C03630=1120.994,-41.227,-48.761,179.607,5.616,149.108
C03631=1120.989,-40.977,-48.773,179.608,5.621,149.109
C03632=1120.983,-40.727,-48.785,179.609,5.626,149.109
C03633=1120.979,-40.477,-48.796,179.611,5.631,149.110
C03634=1120.973,-40.227,-48.808,179.612,5.637,149.111
C03635=1120.969,-39.978,-48.819,179.613,5.642,149.112
C03636=1120.963,-39.729,-48.831,179.614,5.647,149.113
C03637=1120.957,-39.479,-48.843,179.615,5.652,149.113
C03638=1120.952,-39.229,-48.854,179.616,5.658,149.114
C03639=1120.947,-38.979,-48.866,179.618,5.663,149.115
C03640=1120.942,-38.729,-48.878,179.618,5.668,149.116
C03641=1120.937,-38.480,-48.890,179.620,5.673,149.116
C03642=1120.932,-38.230,-48.902,179.620,5.677,149.117
C03643=1120.926,-37.980,-48.914,179.622,5.683,149.118
C03644=1120.921,-37.731,-48.925,179.622,5.687,149.119
C03645=1120.916,-37.481,-48.936,179.624,5.692,149.120
C03646=1120.910,-37.231,-48.948,179.624,5.697,149.120
C03647=1120.905,-36.982,-48.961,179.625,5.702,149.121
C03648=1120.900,-36.733,-48.972,179.626,5.707,149.122
C03649=1120.895,-36.483,-48.984,179.627,5.712,149.123
C03650=1120.889,-36.233,-48.996,179.628,5.716,149.124
C03651=1120.884,-35.983,-49.009,179.628,5.721,149.125
C03652=1120.880,-35.734,-49.020,179.629,5.725,149.125
C03653=1120.874,-35.484,-49.032,179.629,5.730,149.126
C03654=1120.869,-35.234,-49.044,179.630,5.736,149.127
C03655=1120.864,-34.984,-49.056,179.631,5.740,149.128
C03656=1120.858,-34.735,-49.068,179.631,5.744,149.129
C03657=1120.854,-34.485,-49.079,179.632,5.749,149.129
C03658=1120.848,-34.270,-49.090,179.633,5.753,149.130
C03659=1120.844,-34.055,-49.100,179.633,5.757,149.131
C03660=1120.840,-33.840,-49.110,179.633,5.761,149.132
C03661=1120.835,-33.624,-49.121,179.634,5.765,149.132
C03662=1120.831,-33.409,-49.131,179.634,5.768,149.133
C03663=1120.826,-33.194,-49.142,179.634,5.772,149.134
C03664=1120.822,-32.979,-49.152,179.634,5.776,149.135
C03665=1120.817,-32.763,-49.163,179.635,5.779,149.135
C03666=1120.813,-32.514,-49.175,179.635,5.784,149.136
C03667=1120.807,-32.264,-49.186,179.635,5.788,149.137
C03668=1120.802,-32.015,-49.199,179.635,5.793,149.138
C03669=1120.797,-31.765,-49.211,179.635,5.797,149.139
C03670=1120.791,-31.515,-49.223,179.636,5.802,149.140
C03671=1120.786,-31.266,-49.235,179.635,5.806,149.141
C03672=1120.781,-31.016,-49.247,179.636,5.811,149.142
C03673=1120.776,-30.767,-49.259,179.635,5.815,149.143
C03674=1120.771,-30.517,-49.271,179.635,5.819,149.144
C03675=1120.766,-30.268,-49.284,179.635,5.822,149.145
C03676=1120.760,-30.018,-49.296,179.636,5.827,149.146
C03677=1120.755,-29.768,-49.308,179.635,5.832,149.147
C03678=1120.750,-29.518,-49.320,179.635,5.835,149.148
C03679=1120.745,-29.269,-49.333,179.634,5.840,149.149
C03680=1120.739,-29.019,-49.345,179.634,5.844,149.150
C03681=1120.734,-28.769,-49.357,179.634,5.848,149.150
C03682=1120.729,-28.520,-49.369,179.633,5.852,149.152
C03683=1120.724,-28.270,-49.380,179.633,5.856,149.153
C03684=1120.719,-28.021,-49.393,179.633,5.860,149.154
C03685=1120.714,-27.771,-49.406,179.632,5.865,149.155
C03686=1120.709,-27.521,-49.418,179.632,5.869,149.156
C03687=1120.704,-27.272,-49.431,179.631,5.873,149.157
C03688=1120.698,-27.022,-49.442,179.631,5.877,149.158
C03689=1120.693,-26.773,-49.455,179.630,5.882,149.159
C03690=1120.688,-26.523,-49.467,179.630,5.885,149.160
C03691=1120.683,-26.273,-49.479,179.629,5.889,149.161
C03692=1120.677,-26.023,-49.491,179.628,5.893,149.162
C03693=1120.672,-25.774,-49.504,179.628,5.898,149.163
C03694=1120.667,-25.524,-49.516,179.628,5.903,149.164
C03695=1120.662,-25.275,-49.528,179.629,5.908,149.165
C03696=1120.656,-25.025,-49.541,179.629,5.913,149.166
C03697=1120.652,-24.775,-49.553,179.630,5.917,149.167
C03698=1120.647,-24.525,-49.566,179.631,5.923,149.168
C03699=1120.641,-24.276,-49.578,179.632,5.927,149.169
C03700=1120.636,-24.026,-49.590,179.632,5.932,149.169
C03701=1120.631,-23.777,-49.603,179.633,5.937,149.170
C03702=1120.625,-23.527,-49.615,179.634,5.942,149.171
C03703=1120.620,-23.278,-49.627,179.634,5.947,149.172
C03704=1120.615,-23.028,-49.640,179.635,5.952,149.173
C03705=1120.610,-22.778,-49.652,179.635,5.957,149.174
C03706=1120.605,-22.528,-49.665,179.636,5.961,149.175
C03707=1120.600,-22.279,-49.678,179.637,5.966,149.175
C03708=1120.595,-22.029,-49.689,179.638,5.971,149.176
C03709=1120.590,-21.780,-49.702,179.638,5.976,149.177
C03710=1120.584,-21.530,-49.715,179.639,5.981,149.178
C03711=1120.578,-21.280,-49.727,179.639,5.985,149.179
C03712=1120.574,-21.030,-49.740,179.640,5.990,149.180
C03713=1120.569,-20.781,-49.753,179.641,5.994,149.181
C03714=1120.564,-20.566,-49.763,179.641,5.999,149.182
C03715=1120.560,-20.351,-49.774,179.642,6.003,149.182
C03716=1120.555,-20.136,-49.785,179.643,6.007,149.183
C03717=1120.551,-19.921,-49.796,179.643,6.012,149.184
C03718=1120.546,-19.705,-49.807,179.643,6.015,149.184
C03719=1120.542,-19.491,-49.818,179.644,6.020,149.185
C03720=1120.538,-19.275,-49.828,179.645,6.023,149.186
C03721=1120.533,-19.060,-49.839,179.645,6.028,149.187
C03722=1120.528,-18.811,-49.852,179.646,6.032,149.187
C03723=1120.523,-18.562,-49.864,179.647,6.037,149.188
C03724=1120.517,-18.311,-49.878,179.647,6.042,149.189
C03725=1120.512,-18.062,-49.890,179.648,6.047,149.190
C03726=1120.507,-17.813,-49.903,179.648,6.051,149.191
C03727=1120.502,-17.563,-49.915,179.649,6.056,149.192
C03728=1120.498,-17.313,-49.928,179.650,6.060,149.192
C03729=1120.491,-17.063,-49.941,179.650,6.065,149.193
C03730=1120.486,-16.814,-49.954,179.651,6.070,149.194
C03731=1120.481,-16.564,-49.966,179.652,6.075,149.195
C03732=1120.477,-16.314,-49.979,179.653,6.080,149.196
C03733=1120.471,-16.065,-49.992,179.653,6.084,149.197
C03734=1120.466,-15.815,-50.005,179.654,6.089,149.198
C03735=1120.460,-15.566,-50.018,179.655,6.093,149.198
C03736=1120.456,-15.316,-50.030,179.655,6.098,149.199
C03737=1120.450,-15.066,-50.044,179.656,6.103,149.200
C03738=1120.445,-14.817,-50.056,179.656,6.108,149.201
C03739=1120.440,-14.567,-50.069,179.657,6.112,149.202
C03740=1120.435,-14.318,-50.082,179.658,6.117,149.202
C03741=1120.429,-14.068,-50.095,179.658,6.121,149.203
C03742=1120.425,-13.818,-50.108,179.659,6.126,149.204
C03743=1120.420,-13.569,-50.121,179.660,6.131,149.205
C03744=1120.414,-13.319,-50.134,179.660,6.135,149.206
C03745=1120.409,-13.069,-50.147,179.661,6.140,149.207
C03746=1120.404,-12.820,-50.159,179.662,6.144,149.207
C03747=1120.398,-12.570,-50.173,179.662,6.149,149.208
C03748=1120.394,-12.320,-50.186,179.663,6.154,149.209
C03749=1120.389,-12.071,-50.199,179.664,6.158,149.210
C03750=1120.383,-11.822,-50.212,179.664,6.163,149.211
C03751=1120.379,-11.572,-50.225,179.665,6.168,149.212
C03752=1120.374,-11.323,-50.238,179.666,6.172,149.212
C03753=1120.368,-11.073,-50.251,179.666,6.177,149.213
C03754=1120.363,-10.823,-50.264,179.667,6.181,149.214
C03755=1120.358,-10.574,-50.276,179.667,6.186,149.215
C03756=1120.353,-10.324,-50.291,179.668,6.190,149.216
C03757=1120.348,-10.075,-50.303,179.669,6.195,149.216
C03758=1120.342,-9.825,-50.316,179.669,6.200,149.217
C03759=1120.338,-9.575,-50.329,179.670,6.204,149.218
C03760=1120.332,-9.326,-50.342,179.671,6.209,149.219
C03761=1120.327,-9.075,-50.356,179.671,6.214,149.220
C03762=1120.322,-8.827,-50.369,179.672,6.217,149.220
C03763=1120.317,-8.577,-50.382,179.672,6.222,149.221
C03764=1120.312,-8.327,-50.395,179.673,6.227,149.222
C03765=1120.306,-8.077,-50.408,179.674,6.231,149.223
C03766=1120.302,-7.828,-50.422,179.674,6.236,149.224
C03767=1120.296,-7.578,-50.435,179.675,6.240,149.225
C03768=1120.291,-7.329,-50.448,179.676,6.245,149.225
C03769=1120.286,-7.079,-50.462,179.676,6.250,149.226
C03770=1120.282,-6.864,-50.472,179.676,6.253,149.227
C03771=1120.277,-6.649,-50.484,179.677,6.257,149.228
C03772=1120.273,-6.434,-50.495,179.677,6.261,149.228
C03773=1120.269,-6.219,-50.507,179.678,6.266,149.229
C03774=1120.264,-6.004,-50.518,179.679,6.269,149.230
C03775=1120.260,-5.789,-50.530,179.679,6.273,149.230
C03776=1120.255,-5.574,-50.541,179.680,6.277,149.231
C03777=1120.251,-5.360,-50.553,179.680,6.281,149.232
C03778=1120.245,-5.109,-50.566,179.681,6.285,149.233
C03779=1120.241,-4.861,-50.580,179.682,6.290,149.234
C03780=1120.235,-4.610,-50.593,179.682,6.295,149.234
C03781=1120.231,-4.362,-50.606,179.683,6.299,149.235
C03782=1120.225,-4.111,-50.620,179.684,6.304,149.236
C03783=1120.219,-3.862,-50.633,179.683,6.308,149.237
C03784=1120.215,-3.612,-50.647,179.684,6.312,149.238
C03785=1120.209,-3.363,-50.660,179.685,6.317,149.238
C03786=1120.205,-3.113,-50.674,179.685,6.322,149.239
C03787=1120.199,-2.864,-50.687,179.686,6.326,149.240
C03788=1120.194,-2.614,-50.701,179.687,6.331,149.241
C03789=1120.189,-2.365,-50.714,179.688,6.335,149.242
C03790=1120.184,-2.115,-50.728,179.688,6.340,149.243
C03791=1120.179,-1.865,-50.741,179.689,6.344,149.243
C03792=1120.174,-1.616,-50.755,179.689,6.348,149.244
C03793=1120.169,-1.365,-50.769,179.690,6.353,149.245
C03794=1120.164,-1.117,-50.782,179.690,6.358,149.246
C03795=1120.159,-0.866,-50.795,179.691,6.362,149.247
C03796=1120.153,-0.617,-50.809,179.692,6.367,149.247
C03797=1120.149,-0.367,-50.822,179.692,6.372,149.248
C03798=1120.143,-0.118,-50.836,179.693,6.376,149.249
C03799=1120.138,0.132,-50.850,179.693,6.380,149.250
C03800=1120.133,0.381,-50.863,179.694,6.385,149.251
C03801=1120.128,0.631,-50.877,179.694,6.389,149.252
C03802=1120.123,0.881,-50.891,179.695,6.394,149.252
C03803=1120.118,1.129,-50.904,179.696,6.398,149.253
C03804=1120.113,1.380,-50.918,179.696,6.403,149.254
C03805=1120.107,1.629,-50.932,179.697,6.408,149.255
C03806=1120.102,1.879,-50.945,179.698,6.412,149.256
C03807=1120.098,2.128,-50.959,179.698,6.416,149.257
C03808=1120.092,2.377,-50.973,179.698,6.421,149.257
C03809=1120.087,2.628,-50.986,179.699,6.425,149.258
C03810=1120.082,2.877,-51.000,179.699,6.430,149.259
C03811=1120.077,3.126,-51.014,179.700,6.434,149.260
C03812=1120.072,3.377,-51.028,179.701,6.439,149.261
C03813=1120.066,3.626,-51.042,179.701,6.443,149.262
C03814=1120.062,3.875,-51.055,179.701,6.448,149.263
C03815=1120.057,4.125,-51.069,179.702,6.453,149.263
C03816=1120.051,4.374,-51.083,179.703,6.457,149.264
C03817=1120.046,4.624,-51.097,179.703,6.462,149.265
C03818=1120.041,4.874,-51.111,179.704,6.466,149.266
C03819=1120.036,5.123,-51.124,179.704,6.471,149.267
C03820=1120.031,5.373,-51.138,179.704,6.475,149.268
C03821=1120.026,5.622,-51.152,179.705,6.480,149.268
C03822=1120.021,5.871,-51.166,179.706,6.484,149.269
C03823=1120.016,6.121,-51.181,179.706,6.489,149.270
C03824=1120.011,6.372,-51.194,179.707,6.493,149.271
C03825=1120.006,6.620,-51.207,179.707,6.498,149.272
C03826=1120.001,6.835,-51.220,179.708,6.502,149.272
C03827=1119.997,7.050,-51.232,179.708,6.506,149.273
C03828=1119.992,7.265,-51.243,179.708,6.509,149.274
C03829=1119.988,7.480,-51.256,179.709,6.513,149.275
C03830=1119.983,7.695,-51.268,179.709,6.517,149.276
C03831=1119.980,7.910,-51.280,179.710,6.521,149.276
C03832=1119.975,8.124,-51.292,179.711,6.525,149.277
C03833=1119.971,8.340,-51.303,179.711,6.529,149.278
C03834=1119.966,8.589,-51.318,179.711,6.534,149.279
C03835=1119.961,8.839,-51.332,179.712,6.538,149.279
C03836=1119.955,9.088,-51.346,179.713,6.543,149.280
C03837=1119.950,9.338,-51.360,179.713,6.548,149.281
C03838=1119.945,9.588,-51.375,179.714,6.552,149.282
C03839=1119.940,9.837,-51.388,179.715,6.557,149.283
C03840=1119.935,10.086,-51.403,179.715,6.561,149.283
C03841=1119.930,10.336,-51.417,179.716,6.566,149.284
C03842=1119.925,10.586,-51.431,179.717,6.570,149.285
C03843=1119.919,10.835,-51.445,179.718,6.576,149.286
C03844=1119.914,11.084,-51.459,179.719,6.581,149.287
C03845=1119.909,11.334,-51.474,179.720,6.585,149.287
C03846=1119.904,11.584,-51.488,179.720,6.590,149.288
C03847=1119.899,11.833,-51.502,179.721,6.594,149.289
C03848=1119.894,12.082,-51.516,179.722,6.599,149.290
C03849=1119.889,12.332,-51.530,179.722,6.603,149.291
C03850=1119.884,12.582,-51.545,179.723,6.608,149.292
C03851=1119.879,12.832,-51.559,179.724,6.613,149.292
C03852=1119.873,13.081,-51.573,179.724,6.617,149.293
C03853=1119.869,13.330,-51.587,179.725,6.622,149.294
C03854=1119.864,13.580,-51.601,179.726,6.626,149.295
C03855=1119.859,13.830,-51.616,179.727,6.631,149.295
C03856=1119.854,14.079,-51.630,179.728,6.635,149.296
C03857=1119.849,14.329,-51.644,179.728,6.640,149.297
C03858=1119.843,14.578,-51.658,179.729,6.644,149.298
C03859=1119.838,14.828,-51.673,179.730,6.649,149.299
C03860=1119.834,15.077,-51.687,179.731,6.653,149.299
C03861=1119.829,15.327,-51.702,179.731,6.658,149.300
C03862=1119.824,15.576,-51.716,179.732,6.662,149.301
C03863=1119.819,15.826,-51.730,179.733,6.667,149.302
C03864=1119.813,16.075,-51.744,179.734,6.671,149.302
C03865=1119.808,16.325,-51.759,179.735,6.676,149.303
C03866=1119.803,16.574,-51.774,179.736,6.680,149.304
C03867=1119.798,16.824,-51.788,179.736,6.685,149.305
C03868=1119.793,17.074,-51.803,179.737,6.689,149.305
C03869=1119.788,17.323,-51.817,179.738,6.694,149.306
C03870=1119.783,17.572,-51.832,179.739,6.699,149.307
C03871=1119.778,17.822,-51.846,179.739,6.703,149.308
C03872=1119.773,18.071,-51.860,179.740,6.708,149.308
C03873=1119.767,18.321,-51.875,179.741,6.712,149.309
C03874=1119.762,18.570,-51.890,179.742,6.717,149.310
C03875=1119.757,18.820,-51.904,179.743,6.721,149.311
C03876=1119.753,19.070,-51.919,179.744,6.726,149.311
C03877=1119.748,19.319,-51.933,179.745,6.730,149.312
C03878=1119.742,19.569,-51.948,179.746,6.734,149.313
C03879=1119.737,19.819,-51.963,179.746,6.739,149.314
C03880=1119.732,20.068,-51.977,179.747,6.743,149.314
C03881=1119.728,20.317,-51.992,179.748,6.748,149.315
C03882=1119.723,20.532,-52.005,179.749,6.751,149.316
C03883=1119.719,20.747,-52.017,179.750,6.755,149.316
C03884=1119.714,20.961,-52.030,179.750,6.759,149.317
C03885=1119.710,21.176,-52.042,179.751,6.763,149.318
C03886=1119.705,21.391,-52.055,179.752,6.767,149.318
C03887=1119.701,21.606,-52.068,179.752,6.770,149.319
C03888=1119.697,21.821,-52.080,179.754,6.774,149.319
C03889=1119.692,22.036,-52.093,179.754,6.778,149.320
C03890=1119.687,22.285,-52.108,179.755,6.783,149.321
C03891=1119.683,22.535,-52.122,179.756,6.787,149.322
C03892=1119.677,22.785,-52.137,179.757,6.791,149.322
C03893=1119.672,23.034,-52.152,179.758,6.795,149.323
C03894=1119.667,23.284,-52.166,179.758,6.800,149.324
C03895=1119.663,23.533,-52.181,179.759,6.804,149.324
C03896=1119.657,23.783,-52.196,179.760,6.809,149.325
C03897=1119.652,24.032,-52.211,179.762,6.813,149.326
C03898=1119.647,24.281,-52.226,179.762,6.818,149.327
C03899=1119.642,24.531,-52.241,179.763,6.822,149.327
C03900=1119.637,24.781,-52.255,179.764,6.826,149.328
C03901=1119.632,25.030,-52.270,179.765,6.831,149.329
C03902=1119.627,25.280,-52.285,179.766,6.835,149.329
C03903=1119.622,25.529,-52.300,179.767,6.840,149.330
C03904=1119.617,25.778,-52.316,179.768,6.844,149.331
C03905=1119.612,26.028,-52.330,179.769,6.848,149.331
C03906=1119.607,26.277,-52.345,179.770,6.853,149.332
C03907=1119.601,26.527,-52.360,179.771,6.857,149.333
C03908=1119.597,26.776,-52.375,179.772,6.862,149.334
C03909=1119.591,27.026,-52.391,179.772,6.865,149.334
C03910=1119.587,27.276,-52.405,179.773,6.870,149.335
C03911=1119.582,27.525,-52.420,179.774,6.874,149.335
C03912=1119.577,27.774,-52.436,179.775,6.878,149.336
C03913=1119.572,28.024,-52.450,179.776,6.883,149.337
C03914=1119.566,28.274,-52.466,179.777,6.887,149.337
C03915=1119.562,28.523,-52.481,179.778,6.892,149.338
C03916=1119.556,28.773,-52.496,179.779,6.896,149.339
C03917=1119.551,29.022,-52.511,179.780,6.900,149.340
C03918=1119.546,29.271,-52.526,179.781,6.904,149.340
C03919=1119.541,29.521,-52.540,179.782,6.909,149.341
C03920=1119.536,29.770,-52.556,179.783,6.913,149.342
C03921=1119.532,30.020,-52.571,179.784,6.917,149.342
C03922=1119.526,30.269,-52.587,179.785,6.922,149.343
C03923=1119.521,30.519,-52.601,179.786,6.926,149.344
C03924=1119.516,30.769,-52.617,179.787,6.930,149.344
C03925=1119.511,31.018,-52.632,179.789,6.935,149.345
C03926=1119.506,31.267,-52.647,179.789,6.938,149.345
C03927=1119.501,31.517,-52.662,179.790,6.943,149.346
C03928=1119.496,31.767,-52.678,179.791,6.947,149.347
C03929=1119.492,32.016,-52.693,179.792,6.951,149.347
C03930=1119.486,32.265,-52.708,179.793,6.955,149.348
C03931=1119.482,32.514,-52.723,179.794,6.960,149.349
C03932=1119.476,32.764,-52.739,179.795,6.964,149.349
C03933=1119.471,33.013,-52.754,179.796,6.968,149.350
C03934=1119.466,33.264,-52.769,179.797,6.973,149.351
C03935=1119.461,33.513,-52.785,179.799,6.977,149.351
C03936=1119.456,33.762,-52.800,179.800,6.981,149.352
C03937=1119.451,34.012,-52.815,179.801,6.986,149.353
C03938=1119.446,34.227,-52.828,179.801,6.989,149.353
C03939=1119.442,34.441,-52.842,179.802,6.992,149.354
C03940=1119.437,34.656,-52.855,179.803,6.997,149.354
C03941=1119.433,34.870,-52.869,179.804,7.000,149.355
C03942=1119.430,35.085,-52.881,179.805,7.004,149.355
C03943=1119.426,35.300,-52.895,179.806,7.007,149.356
C03944=1119.421,35.515,-52.908,179.806,7.011,149.357
C03945=1119.417,35.729,-52.922,179.808,7.015,149.357
C03946=1119.411,35.979,-52.937,179.809,7.019,149.358
C03947=1119.406,36.228,-52.952,179.809,7.022,149.358
C03948=1119.402,36.478,-52.968,179.811,7.027,149.359
C03949=1119.397,36.727,-52.984,179.812,7.031,149.360
C03950=1119.391,36.977,-52.999,179.813,7.035,149.360
C03951=1119.386,37.226,-53.014,179.814,7.040,149.361
C03952=1119.382,37.476,-53.030,179.815,7.044,149.361
C03953=1119.376,37.725,-53.046,179.816,7.048,149.362
C03954=1119.372,37.974,-53.061,179.817,7.052,149.363
C03955=1119.366,38.224,-53.077,179.818,7.057,149.363
C03956=1119.361,38.474,-53.093,179.820,7.061,149.364
C03957=1119.356,38.723,-53.108,179.821,7.065,149.365
C03958=1119.351,38.972,-53.123,179.822,7.069,149.365
C03959=1119.347,39.222,-53.139,179.823,7.073,149.366
C03960=1119.341,39.472,-53.155,179.824,7.077,149.366
C03961=1119.336,39.721,-53.170,179.825,7.081,149.367
C03962=1119.332,39.970,-53.186,179.826,7.086,149.368
C03963=1119.327,40.220,-53.202,179.827,7.090,149.368
C03964=1119.321,40.469,-53.217,179.828,7.094,149.369
C03965=1119.316,40.718,-53.233,179.830,7.098,149.369
C03966=1119.311,40.969,-53.249,179.831,7.102,149.370
C03967=1119.306,41.217,-53.265,179.832,7.107,149.371
C03968=1119.301,41.466,-53.280,179.833,7.111,149.371
C03969=1119.297,41.717,-53.296,179.834,7.114,149.372
C03970=1119.291,41.966,-53.312,179.835,7.118,149.372
C03971=1119.286,42.215,-53.327,179.836,7.123,149.373
C03972=1119.281,42.465,-53.344,179.837,7.127,149.374
C03973=1119.276,42.714,-53.360,179.838,7.131,149.374
C03974=1119.271,42.963,-53.375,179.840,7.135,149.375
C03975=1119.267,43.213,-53.391,179.841,7.140,149.375
C03976=1119.262,43.462,-53.407,179.842,7.144,149.376
C03977=1119.257,43.712,-53.423,179.843,7.148,149.376
C03978=1119.251,43.962,-53.439,179.844,7.152,149.377
C03979=1119.246,44.211,-53.455,179.845,7.156,149.378
C03980=1119.241,44.461,-53.471,179.846,7.159,149.378
C03981=1119.236,44.710,-53.486,179.847,7.164,149.379
C03982=1119.232,44.960,-53.503,179.848,7.168,149.379
C03983=1119.226,45.209,-53.519,179.850,7.172,149.380
C03984=1119.222,45.457,-53.534,179.851,7.176,149.381
C03985=1119.217,45.707,-53.550,179.852,7.181,149.381
C03986=1119.212,45.957,-53.566,179.853,7.185,149.382
C03987=1119.207,46.206,-53.583,179.855,7.189,149.382
C03988=1119.202,46.456,-53.598,179.856,7.193,149.383
C03989=1119.197,46.705,-53.615,179.857,7.197,149.384
C03990=1119.192,46.955,-53.630,179.858,7.201,149.384
C03991=1119.187,47.204,-53.646,179.859,7.205,149.385
C03992=1119.182,47.454,-53.663,179.861,7.209,149.385
C03993=1119.177,47.703,-53.678,179.862,7.213,149.386
C03994=1119.173,47.918,-53.692,179.863,7.216,149.386
C03995=1119.168,48.133,-53.707,179.864,7.221,149.387
C03996=1119.164,48.347,-53.720,179.865,7.224,149.387
C03997=1119.160,48.562,-53.734,179.866,7.228,149.388
C03998=1119.156,48.776,-53.748,179.867,7.231,149.388
C03999=1119.151,48.991,-53.762,179.867,7.234,149.389
C04000=1119.147,49.205,-53.776,179.869,7.238,149.389
C04001=1119.143,49.420,-53.790,179.870,7.241,149.390
C04002=1119.138,49.669,-53.806,179.871,7.246,149.390
C04003=1119.133,49.919,-53.822,179.873,7.249,149.391
C04004=1119.128,50.168,-53.839,179.874,7.254,149.391
C04005=1119.123,50.418,-53.855,179.875,7.258,149.392
C04006=1119.118,50.667,-53.871,179.876,7.261,149.392
C04007=1119.113,50.916,-53.888,179.877,7.265,149.393
C04008=1119.108,51.166,-53.903,179.878,7.269,149.394
C04009=1119.104,51.415,-53.920,179.879,7.274,149.394
C04010=1119.098,51.665,-53.936,179.881,7.278,149.395
C04011=1119.093,51.914,-53.953,179.882,7.282,149.395
C04012=1119.088,52.163,-53.969,179.884,7.286,149.396
C04013=1119.083,52.413,-53.985,179.885,7.290,149.396
C04014=1119.079,52.663,-54.002,179.886,7.294,149.397
C04015=1119.074,52.912,-54.018,179.887,7.298,149.397
C04016=1119.069,53.162,-54.034,179.888,7.302,149.398
C04017=1119.063,53.411,-54.051,179.889,7.306,149.398
C04018=1119.058,53.660,-54.068,179.890,7.310,149.399
C04019=1119.053,53.909,-54.084,179.892,7.314,149.400
C04020=1119.049,54.159,-54.100,179.893,7.318,149.400
C04021=1119.044,54.409,-54.116,179.895,7.322,149.401
C04022=1119.038,54.658,-54.133,179.896,7.326,149.401
C04023=1119.034,54.907,-54.150,179.897,7.330,149.402
C04024=1119.028,55.157,-54.166,179.898,7.335,149.402
C04025=1119.024,55.406,-54.182,179.899,7.338,149.403
C04026=1119.019,55.656,-54.199,179.900,7.342,149.403
C04027=1119.014,55.905,-54.216,179.902,7.346,149.404
C04028=1119.009,56.154,-54.233,179.903,7.350,149.404
C04029=1119.004,56.403,-54.249,179.905,7.354,149.405
C04030=1118.999,56.653,-54.265,179.906,7.359,149.406
C04031=1118.994,56.903,-54.282,179.907,7.362,149.406
C04032=1118.989,57.152,-54.298,179.908,7.367,149.407
C04033=1118.984,57.401,-54.315,179.910,7.371,149.407
C04034=1118.979,57.651,-54.332,179.911,7.375,149.408
C04035=1118.974,57.900,-54.349,179.912,7.378,149.408
C04036=1118.970,58.149,-54.365,179.914,7.382,149.409
C04037=1118.964,58.399,-54.383,179.915,7.386,149.409
C04038=1118.959,58.648,-54.399,179.916,7.390,149.410
C04039=1118.955,58.897,-54.415,179.917,7.394,149.410
C04040=1118.949,59.148,-54.432,179.919,7.398,149.411
C04041=1118.944,59.396,-54.448,179.920,7.403,149.411
C04042=1118.940,59.646,-54.465,179.922,7.407,149.412
C04043=1118.935,59.896,-54.482,179.923,7.411,149.412
C04044=1118.930,60.145,-54.499,179.924,7.415,149.413
C04045=1118.925,60.394,-54.515,179.925,7.418,149.413
C04046=1118.920,60.644,-54.532,179.926,7.422,149.414
C04047=1118.915,60.893,-54.549,179.928,7.426,149.414
C04048=1118.910,61.142,-54.566,179.929,7.430,149.415
C04049=1118.905,61.391,-54.583,179.931,7.434,149.415
C04050=1118.901,61.606,-54.597,179.931,7.437,149.416
C04051=1118.897,61.821,-54.612,179.933,7.441,149.416
C04052=1118.893,62.035,-54.626,179.934,7.444,149.417
C04053=1118.888,62.250,-54.641,179.936,7.448,149.417
C04054=1118.884,62.464,-54.655,179.936,7.452,149.418
C04055=1118.880,62.679,-54.670,179.937,7.455,149.418
C04056=1118.876,62.893,-54.684,179.939,7.459,149.419
C04057=1118.871,63.108,-54.699,179.940,7.462,149.419
C04058=1118.867,63.357,-54.716,179.941,7.466,149.420
C04059=1118.861,63.606,-54.733,179.943,7.470,149.420
C04060=1118.857,63.855,-54.750,179.944,7.474,149.421
C04061=1118.852,64.105,-54.767,179.945,7.478,149.421
C04062=1118.847,64.355,-54.784,179.947,7.482,149.422
C04063=1118.841,64.604,-54.801,179.947,7.485,149.422
C04064=1118.837,64.853,-54.818,179.949,7.489,149.423
C04065=1118.832,65.103,-54.836,179.950,7.493,149.423
C04066=1118.828,65.352,-54.852,179.952,7.498,149.424
C04067=1118.822,65.602,-54.869,179.953,7.501,149.424
C04068=1118.818,65.850,-54.886,179.955,7.505,149.425
C04069=1118.812,66.100,-54.904,179.956,7.510,149.425
C04070=1118.807,66.350,-54.921,179.957,7.514,149.426
C04071=1118.803,66.599,-54.938,179.959,7.517,149.426
C04072=1118.798,66.848,-54.956,179.960,7.522,149.427
C04073=1118.793,67.098,-54.972,179.962,7.526,149.427
C04074=1118.787,67.347,-54.989,179.963,7.529,149.428
C04075=1118.783,67.596,-55.007,179.964,7.533,149.428
C04076=1118.778,67.845,-55.024,179.965,7.537,149.429
C04077=1118.773,68.095,-55.041,179.967,7.541,149.429
C04078=1118.769,68.344,-55.059,179.968,7.545,149.430
C04079=1118.763,68.594,-55.076,179.970,7.549,149.430
C04080=1118.759,68.843,-55.092,179.971,7.553,149.431
C04081=1118.753,69.092,-55.110,179.972,7.557,149.431
C04082=1118.748,69.342,-55.127,179.974,7.561,149.432
C04083=1118.744,69.591,-55.144,179.975,7.565,149.432
C04084=1118.739,69.840,-55.162,179.976,7.569,149.433
C04085=1118.734,70.090,-55.179,179.978,7.573,149.433
C04086=1118.729,70.339,-55.197,179.980,7.577,149.434
C04087=1118.724,70.589,-55.214,179.981,7.581,149.434
C04088=1118.719,70.838,-55.232,179.982,7.585,149.435
C04089=1118.715,71.087,-55.249,179.983,7.588,149.435
C04090=1118.710,71.337,-55.267,179.985,7.592,149.436
C04091=1118.704,71.586,-55.283,179.986,7.597,149.436
C04092=1118.700,71.835,-55.301,179.987,7.601,149.437
C04093=1118.695,72.084,-55.318,179.989,7.604,149.437
C04094=1118.690,72.334,-55.336,179.990,7.609,149.438
C04095=1118.685,72.583,-55.353,179.992,7.613,149.438
C04096=1118.680,72.832,-55.371,179.993,7.617,149.439
C04097=1118.675,73.082,-55.388,179.995,7.620,149.439
C04098=1118.670,73.331,-55.406,179.996,7.625,149.440
C04099=1118.665,73.581,-55.423,179.998,7.629,149.440
C04100=1118.661,73.830,-55.441,179.999,7.633,149.440
C04101=1118.656,74.079,-55.459,-179.999,7.636,149.441
C04102=1118.651,74.329,-55.476,-179.998,7.641,149.442
C04103=1118.646,74.578,-55.494,-179.997,7.644,149.442
C04104=1118.641,74.827,-55.512,-179.996,7.648,149.442
C04105=1118.636,75.077,-55.528,-179.994,7.652,149.443
C04106=1118.632,75.291,-55.544,-179.992,7.656,149.443
C04107=1118.628,75.505,-55.559,-179.991,7.659,149.444
C04108=1118.623,75.720,-55.574,-179.990,7.663,149.444
C04109=1118.619,75.935,-55.590,-179.989,7.666,149.445
C04110=1118.615,76.149,-55.605,-179.988,7.669,149.445
C04111=1118.611,76.363,-55.619,-179.986,7.673,149.445
C04112=1118.607,76.578,-55.635,-179.985,7.676,149.446
C04113=1118.602,76.792,-55.650,-179.984,7.680,149.446
C04114=1118.597,77.041,-55.668,-179.983,7.683,149.447
C04115=1118.593,77.290,-55.686,-179.982,7.686,149.447
C04116=1118.588,77.540,-55.704,-179.981,7.691,149.448
C04117=1118.582,77.789,-55.721,-179.980,7.694,149.448
C04118=1118.578,78.039,-55.739,-179.979,7.698,149.449
C04119=1118.573,78.288,-55.757,-179.979,7.702,149.450
C04120=1118.569,78.537,-55.775,-179.977,7.705,149.450
C04121=1118.564,78.787,-55.792,-179.977,7.709,149.451
C04122=1118.559,79.036,-55.810,-179.975,7.713,149.451
C04123=1118.554,79.285,-55.828,-179.975,7.716,149.452
C04124=1118.549,79.535,-55.846,-179.973,7.720,149.452
C04125=1118.544,79.784,-55.864,-179.972,7.724,149.453
C04126=1118.539,80.033,-55.882,-179.971,7.728,149.453
C04127=1118.534,80.283,-55.899,-179.970,7.731,149.454
C04128=1118.529,80.532,-55.917,-179.969,7.735,149.454
C04129=1118.524,80.781,-55.935,-179.968,7.739,149.455
C04130=1118.519,81.030,-55.953,-179.967,7.742,149.456
C04131=1118.515,81.280,-55.971,-179.966,7.746,149.456
C04132=1118.510,81.529,-55.989,-179.965,7.750,149.457
C04133=1118.505,81.778,-56.007,-179.963,7.754,149.457
C04134=1118.500,82.028,-56.025,-179.962,7.757,149.458
C04135=1118.495,82.277,-56.043,-179.961,7.761,149.458
C04136=1118.490,82.526,-56.061,-179.960,7.765,149.459
C04137=1118.485,82.776,-56.079,-179.959,7.769,149.459
C04138=1118.480,83.025,-56.097,-179.958,7.773,149.460
C04139=1118.475,83.274,-56.115,-179.957,7.776,149.460
C04140=1118.471,83.524,-56.133,-179.956,7.780,149.461
C04141=1118.466,83.773,-56.151,-179.954,7.784,149.461
C04142=1118.461,84.022,-56.169,-179.953,7.788,149.462
C04143=1118.456,84.272,-56.187,-179.952,7.791,149.462
C04144=1118.451,84.521,-56.205,-179.951,7.796,149.463
C04145=1118.446,84.770,-56.223,-179.950,7.799,149.464
C04146=1118.442,85.020,-56.241,-179.948,7.803,149.464
C04147=1118.438,85.268,-56.260,-179.947,7.807,149.465
C04148=1118.432,85.518,-56.278,-179.946,7.810,149.465
C04149=1118.427,85.767,-56.296,-179.945,7.814,149.466
C04150=1118.422,86.016,-56.314,-179.943,7.818,149.466
C04151=1118.417,86.265,-56.332,-179.942,7.822,149.467
C04152=1118.413,86.515,-56.351,-179.941,7.826,149.467
C04153=1118.408,86.764,-56.369,-179.940,7.830,149.468
C04154=1118.403,87.014,-56.387,-179.938,7.833,149.468
C04155=1118.398,87.263,-56.405,-179.937,7.838,149.469
C04156=1118.393,87.513,-56.424,-179.936,7.841,149.469
C04157=1118.388,87.761,-56.442,-179.934,7.845,149.470
C04158=1118.384,88.011,-56.460,-179.933,7.849,149.470
C04159=1118.379,88.260,-56.478,-179.932,7.853,149.471
C04160=1118.374,88.509,-56.496,-179.931,7.856,149.471
C04161=1118.369,88.759,-56.515,-179.929,7.860,149.471
C04162=1118.364,88.973,-56.531,-179.928,7.863,149.472
C04163=1118.360,89.187,-56.546,-179.927,7.867,149.472
C04164=1118.356,89.401,-56.562,-179.926,7.870,149.473
C04165=1118.352,89.616,-56.578,-179.925,7.873,149.473
C04166=1118.348,89.830,-56.594,-179.923,7.877,149.474
C04167=1118.344,90.045,-56.609,-179.922,7.880,149.474
C04168=1118.340,90.259,-56.626,-179.921,7.883,149.474
C04169=1118.336,90.474,-56.641,-179.919,7.887,149.475
C04170=1118.331,90.723,-56.660,-179.918,7.890,149.475
C04171=1118.326,90.972,-56.678,-179.917,7.894,149.476
C04172=1118.321,91.221,-56.696,-179.915,7.898,149.476
C04173=1118.316,91.471,-56.716,-179.914,7.902,149.477
C04174=1118.311,91.720,-56.734,-179.912,7.906,149.477
C04175=1118.307,91.969,-56.752,-179.911,7.910,149.478
C04176=1118.302,92.219,-56.771,-179.909,7.914,149.478
C04177=1118.297,92.468,-56.789,-179.908,7.918,149.479
C04178=1118.292,92.717,-56.807,-179.907,7.921,149.479
C04179=1118.287,92.965,-56.826,-179.905,7.925,149.479
C04180=1118.282,93.216,-56.845,-179.904,7.929,149.480
C04181=1118.277,93.465,-56.863,-179.902,7.933,149.480
C04182=1118.273,93.713,-56.882,-179.900,7.937,149.481
C04183=1118.268,93.964,-56.901,-179.899,7.940,149.481
C04184=1118.263,94.212,-56.919,-179.897,7.944,149.482
C04185=1118.258,94.462,-56.938,-179.896,7.948,149.482
C04186=1118.253,94.711,-56.957,-179.894,7.952,149.482
C04187=1118.249,94.960,-56.975,-179.892,7.956,149.483
C04188=1118.244,95.210,-56.994,-179.891,7.960,149.483
C04189=1118.239,95.459,-57.012,-179.889,7.964,149.484
C04190=1118.234,95.707,-57.031,-179.888,7.968,149.484
C04191=1118.229,95.957,-57.050,-179.886,7.972,149.485
C04192=1118.225,96.206,-57.069,-179.884,7.975,149.485
C04193=1118.219,96.456,-57.087,-179.883,7.979,149.485
C04194=1118.215,96.705,-57.106,-179.881,7.983,149.486
C04195=1118.209,96.954,-57.125,-179.880,7.987,149.486
C04196=1118.205,97.204,-57.144,-179.878,7.991,149.487
C04197=1118.200,97.453,-57.162,-179.876,7.995,149.487
C04198=1118.195,97.702,-57.181,-179.875,7.999,149.488
C04199=1118.191,97.951,-57.200,-179.873,8.002,149.488
C04200=1118.185,98.200,-57.219,-179.871,8.006,149.488
C04201=1118.181,98.450,-57.238,-179.870,8.010,149.489
C04202=1118.176,98.699,-57.257,-179.868,8.014,149.489
C04203=1118.172,98.948,-57.276,-179.866,8.018,149.490
C04204=1118.166,99.197,-57.295,-179.864,8.021,149.490
C04205=1118.162,99.447,-57.313,-179.863,8.025,149.490
C04206=1118.157,99.696,-57.333,-179.861,8.029,149.491
C04207=1118.152,99.944,-57.351,-179.859,8.034,149.491
C04208=1118.147,100.195,-57.370,-179.857,8.037,149.491
C04209=1118.143,100.443,-57.389,-179.855,8.041,149.492
C04210=1118.138,100.693,-57.409,-179.854,8.045,149.492
C04211=1118.132,100.942,-57.428,-179.852,8.049,149.493
C04212=1118.128,101.192,-57.446,-179.850,8.052,149.493
C04213=1118.123,101.440,-57.466,-179.848,8.056,149.493
C04214=1118.119,101.690,-57.485,-179.847,8.060,149.494
C04215=1118.113,101.939,-57.504,-179.845,8.064,149.494
C04216=1118.109,102.188,-57.524,-179.842,8.068,149.494
C04217=1118.104,102.437,-57.541,-179.840,8.072,149.495
C04218=1118.099,102.652,-57.558,-179.839,8.075,149.495
C04219=1118.095,102.866,-57.574,-179.837,8.079,149.495
C04220=1118.092,103.080,-57.592,-179.836,8.081,149.495
C04221=1118.088,103.294,-57.608,-179.834,8.085,149.496
C04222=1118.083,103.509,-57.625,-179.832,8.089,149.496
C04223=1118.080,103.723,-57.641,-179.831,8.091,149.496
C04224=1118.075,103.937,-57.658,-179.829,8.095,149.497
C04225=1118.071,104.151,-57.674,-179.828,8.098,149.497
C04226=1118.066,104.400,-57.693,-179.825,8.102,149.497
C04227=1118.061,104.650,-57.713,-179.824,8.106,149.498
C04228=1118.057,104.899,-57.732,-179.821,8.110,149.498
C04229=1118.052,105.148,-57.751,-179.820,8.114,149.498
C04230=1118.047,105.398,-57.771,-179.818,8.117,149.499
C04231=1118.042,105.646,-57.789,-179.816,8.121,149.499
C04232=1118.038,105.896,-57.809,-179.813,8.125,149.499
C04233=1118.032,106.145,-57.828,-179.811,8.129,149.499
C04234=1118.028,106.394,-57.848,-179.810,8.133,149.500
C04235=1118.024,106.643,-57.867,-179.808,8.136,149.500
C04236=1118.018,106.892,-57.886,-179.805,8.140,149.500
C04237=1118.013,107.142,-57.906,-179.803,8.144,149.501
C04238=1118.009,107.391,-57.926,-179.801,8.148,149.501
C04239=1118.004,107.640,-57.944,-179.799,8.151,149.501
C04240=1117.999,107.889,-57.964,-179.797,8.156,149.501
C04241=1117.994,108.138,-57.983,-179.795,8.159,149.502
C04242=1117.989,108.388,-58.003,-179.793,8.163,149.502
C04243=1117.985,108.638,-58.023,-179.791,8.166,149.502
C04244=1117.980,108.885,-58.042,-179.788,8.171,149.502
C04245=1117.976,109.135,-58.062,-179.786,8.174,149.503
C04246=1117.971,109.385,-58.081,-179.785,8.178,149.503
C04247=1117.965,109.633,-58.101,-179.783,8.182,149.503
C04248=1117.961,109.883,-58.120,-179.780,8.186,149.504
C04249=1117.956,110.133,-58.140,-179.778,8.189,149.504
C04250=1117.951,110.382,-58.160,-179.776,8.193,149.504
C04251=1117.946,110.630,-58.180,-179.773,8.197,149.504
C04252=1117.942,110.880,-58.199,-179.771,8.201,149.504
C04253=1117.937,111.129,-58.218,-179.769,8.204,149.505
C04254=1117.932,111.377,-58.238,-179.767,8.208,149.505
C04255=1117.928,111.627,-58.258,-179.765,8.212,149.505
C04256=1117.923,111.877,-58.278,-179.763,8.215,149.506
C04257=1117.918,112.125,-58.298,-179.762,8.218,149.506
C04258=1117.913,112.374,-58.317,-179.760,8.222,149.506
C04259=1117.908,112.624,-58.337,-179.758,8.225,149.506
C04260=1117.904,112.873,-58.357,-179.756,8.229,149.507
C04261=1117.899,113.122,-58.377,-179.754,8.233,149.507
C04262=1117.894,113.371,-58.396,-179.752,8.236,149.507
C04263=1117.889,113.620,-58.417,-179.751,8.239,149.508
C04264=1117.885,113.870,-58.436,-179.749,8.243,149.508
C04265=1117.879,114.119,-58.456,-179.747,8.246,149.508
C04266=1117.875,114.368,-58.476,-179.745,8.250,149.508
C04267=1117.870,114.617,-58.496,-179.743,8.253,149.509
C04268=1117.866,114.866,-58.516,-179.742,8.256,149.509
C04269=1117.861,115.116,-58.536,-179.740,8.260,149.509
C04270=1117.855,115.461,-58.563,-179.737,8.265,149.510
C04271=1117.848,115.807,-58.591,-179.735,8.269,149.510
C04272=1117.841,116.152,-58.618,-179.732,8.274,149.510
C04273=1117.834,116.498,-58.646,-179.730,8.279,149.511
C04274=1117.828,116.829,-58.673,-179.727,8.283,149.511
C04275=1117.822,117.161,-58.699,-179.725,8.288,149.512
C04276=1117.815,117.493,-58.727,-179.723,8.292,149.512
C04277=1117.809,117.825,-58.753,-179.720,8.297,149.512
C04278=1117.804,118.075,-58.774,-179.719,8.301,149.513
C04279=1117.799,118.324,-58.794,-179.716,8.304,149.513
C04280=1117.795,118.573,-58.814,-179.714,8.307,149.513
C04281=1117.790,118.821,-58.834,-179.713,8.310,149.513
C04282=1117.785,119.071,-58.853,-179.711,8.314,149.514
C04283=1117.780,119.320,-58.874,-179.709,8.318,149.514
C04284=1117.776,119.569,-58.894,-179.707,8.321,149.514
C04285=1117.770,119.819,-58.914,-179.706,8.324,149.514
C04286=1117.766,120.068,-58.935,-179.704,8.328,149.515
C04287=1117.762,120.317,-58.955,-179.702,8.331,149.515
C04288=1117.757,120.566,-58.975,-179.700,8.335,149.515
C04289=1117.752,120.815,-58.995,-179.699,8.337,149.516
C04290=1117.747,121.064,-59.016,-179.697,8.341,149.516
C04291=1117.742,121.313,-59.035,-179.695,8.345,149.516
C04292=1117.737,121.562,-59.056,-179.693,8.348,149.516
C04293=1117.733,121.811,-59.076,-179.691,8.351,149.517
C04294=1117.729,122.060,-59.096,-179.689,8.354,149.517
C04295=1117.723,122.310,-59.117,-179.688,8.358,149.517
C04296=1117.719,122.559,-59.137,-179.686,8.361,149.518
C04297=1117.714,122.808,-59.157,-179.684,8.365,149.518
C04298=1117.709,123.057,-59.178,-179.682,8.368,149.518
C04299=1117.705,123.306,-59.199,-179.681,8.372,149.518
C04300=1117.700,123.556,-59.218,-179.679,8.375,149.519
C04301=1117.695,123.805,-59.239,-179.677,8.378,149.519
C04302=1117.690,124.054,-59.260,-179.675,8.382,149.519
C04303=1117.686,124.303,-59.280,-179.674,8.384,149.519
C04304=1117.681,124.552,-59.301,-179.672,8.388,149.520
C04305=1117.676,124.801,-59.321,-179.670,8.392,149.520
C04306=1117.672,125.050,-59.342,-179.668,8.395,149.520
C04307=1117.667,125.299,-59.362,-179.666,8.398,149.520
C04308=1117.662,125.549,-59.382,-179.665,8.402,149.521
C04309=1117.657,125.798,-59.403,-179.663,8.405,149.521
C04310=1117.653,126.047,-59.423,-179.661,8.408,149.521
C04311=1117.648,126.296,-59.444,-179.659,8.412,149.522
C04312=1117.643,126.545,-59.465,-179.657,8.415,149.522
C04313=1117.639,126.794,-59.485,-179.656,8.418,149.522
C04314=1117.634,127.043,-59.506,-179.654,8.422,149.522
C04315=1117.629,127.292,-59.526,-179.652,8.425,149.523
C04316=1117.624,127.541,-59.547,-179.651,8.428,149.523
C04317=1117.620,127.790,-59.568,-179.649,8.432,149.523
C04318=1117.615,128.040,-59.589,-179.647,8.435,149.524
C04319=1117.610,128.289,-59.609,-179.645,8.438,149.524
C04320=1117.606,128.537,-59.629,-179.644,8.442,149.524
C04321=1117.601,128.787,-59.650,-179.642,8.445,149.524
C04322=1117.596,129.036,-59.671,-179.640,8.448,149.525
C04323=1117.591,129.285,-59.692,-179.638,8.452,149.525
C04324=1117.586,129.534,-59.712,-179.637,8.455,149.525
C04325=1117.582,129.783,-59.734,-179.635,8.458,149.526
C04326=1117.578,129.997,-59.751,-179.634,8.461,149.526
C04327=1117.574,130.211,-59.769,-179.632,8.464,149.526
C04328=1117.570,130.425,-59.787,-179.630,8.467,149.526
C04329=1117.565,130.639,-59.805,-179.629,8.470,149.526
C04330=1117.562,130.853,-59.823,-179.627,8.472,149.527
C04331=1117.557,131.067,-59.841,-179.626,8.475,149.527
C04332=1117.554,131.282,-59.858,-179.625,8.478,149.527
C04333=1117.550,131.495,-59.876,-179.623,8.481,149.528
C04334=1117.545,131.744,-59.897,-179.621,8.484,149.528
C04335=1117.540,131.993,-59.918,-179.619,8.488,149.528
C04336=1117.536,132.243,-59.939,-179.618,8.491,149.528
C04337=1117.530,132.492,-59.960,-179.616,8.495,149.529
C04338=1117.526,132.741,-59.980,-179.614,8.498,149.529
C04339=1117.521,132.990,-60.002,-179.613,8.501,149.529
C04340=1117.517,133.239,-60.023,-179.611,8.505,149.530
C04341=1117.512,133.488,-60.043,-179.609,8.508,149.530
C04342=1117.506,133.737,-60.064,-179.607,8.511,149.530
C04343=1117.503,133.986,-60.086,-179.606,8.515,149.530
C04344=1117.498,134.236,-60.107,-179.604,8.517,149.531
C04345=1117.493,134.484,-60.127,-179.602,8.521,149.531
C04346=1117.488,134.733,-60.149,-179.601,8.525,149.531
C04347=1117.483,134.982,-60.170,-179.599,8.527,149.532
C04348=1117.479,135.231,-60.190,-179.597,8.531,149.532
C04349=1117.475,135.481,-60.212,-179.596,8.535,149.532
C04350=1117.469,135.730,-60.233,-179.594,8.538,149.533
C04351=1117.465,135.979,-60.254,-179.592,8.541,149.533
C04352=1117.460,136.228,-60.275,-179.590,8.545,149.533
C04353=1117.455,136.477,-60.296,-179.589,8.548,149.533
C04354=1117.451,136.726,-60.317,-179.587,8.551,149.534
C04355=1117.446,136.975,-60.339,-179.586,8.554,149.534
C04356=1117.441,137.224,-60.360,-179.584,8.558,149.534
C04357=1117.437,137.473,-60.381,-179.582,8.562,149.535
C04358=1117.432,137.722,-60.402,-179.581,8.564,149.535
C04359=1117.427,137.971,-60.424,-179.579,8.568,149.535
C04360=1117.423,138.220,-60.444,-179.578,8.571,149.536
C04361=1117.418,138.469,-60.466,-179.576,8.574,149.536
C04362=1117.413,138.718,-60.487,-179.574,8.578,149.536
C04363=1117.408,138.968,-60.508,-179.572,8.581,149.537
C04364=1117.404,139.216,-60.529,-179.570,8.584,149.537
C04365=1117.399,139.465,-60.551,-179.569,8.588,149.537
C04366=1117.394,139.714,-60.572,-179.567,8.591,149.537
C04367=1117.390,139.964,-60.594,-179.566,8.595,149.538
C04368=1117.385,140.213,-60.614,-179.564,8.598,149.538
C04369=1117.381,140.461,-60.636,-179.563,8.601,149.539
C04370=1117.376,140.711,-60.657,-179.560,8.605,149.539
C04371=1117.371,140.960,-60.679,-179.559,8.608,149.539
C04372=1117.366,141.209,-60.700,-179.557,8.612,149.539
C04373=1117.362,141.457,-60.721,-179.556,8.614,149.540
C04374=1117.358,141.707,-60.743,-179.554,8.618,149.540
C04375=1117.352,141.956,-60.764,-179.552,8.622,149.540
C04376=1117.348,142.205,-60.786,-179.551,8.625,149.541
C04377=1117.343,142.454,-60.808,-179.549,8.628,149.541
C04378=1117.338,142.703,-60.829,-179.548,8.631,149.541
C04379=1117.334,142.952,-60.850,-179.546,8.635,149.542
C04380=1117.330,143.201,-60.872,-179.544,8.639,149.542
C04381=1117.325,143.450,-60.893,-179.543,8.641,149.542
C04382=1117.320,143.664,-60.912,-179.542,8.644,149.543
C04383=1117.316,143.878,-60.930,-179.540,8.648,149.543
C04384=1117.312,144.092,-60.948,-179.538,8.651,149.543
C04385=1117.309,144.306,-60.967,-179.537,8.654,149.544
C04386=1117.304,144.520,-60.986,-179.536,8.656,149.544
C04387=1117.301,144.734,-61.004,-179.535,8.659,149.544
C04388=1117.297,144.948,-61.023,-179.534,8.662,149.545
C04389=1117.292,145.162,-61.041,-179.532,8.665,149.545
C04390=1117.288,145.411,-61.063,-179.530,8.668,149.545
C04391=1117.283,145.660,-61.084,-179.527,8.673,149.545
C04392=1117.278,145.908,-61.106,-179.525,8.676,149.545
C04393=1117.274,146.158,-61.127,-179.523,8.680,149.546
C04394=1117.269,146.407,-61.149,-179.520,8.684,149.546
C04395=1117.265,146.656,-61.171,-179.518,8.687,149.546
C04396=1117.260,146.905,-61.193,-179.516,8.691,149.546
C04397=1117.255,147.153,-61.214,-179.514,8.695,149.547
C04398=1117.251,147.403,-61.237,-179.511,8.699,149.547
C04399=1117.246,147.651,-61.258,-179.509,8.702,149.547
C04400=1117.242,147.901,-61.280,-179.507,8.706,149.547
C04401=1117.236,148.150,-61.301,-179.505,8.710,149.548
C04402=1117.232,148.399,-61.323,-179.503,8.713,149.548
C04403=1117.227,148.648,-61.345,-179.500,8.717,149.548
C04404=1117.222,148.897,-61.367,-179.498,8.720,149.548
C04405=1117.218,149.146,-61.389,-179.496,8.725,149.549
C04406=1117.212,149.395,-61.411,-179.494,8.728,149.549
C04407=1117.208,149.644,-61.433,-179.491,8.732,149.549
C04408=1117.203,149.893,-61.455,-179.489,8.735,149.549
C04409=1117.199,150.142,-61.477,-179.486,8.739,149.549
C04410=1117.194,150.391,-61.498,-179.484,8.743,149.550
C04411=1117.190,150.640,-61.520,-179.482,8.746,149.550
C04412=1117.185,150.889,-61.542,-179.480,8.749,149.550
C04413=1117.181,151.138,-61.564,-179.478,8.753,149.550
C04414=1117.175,151.387,-61.586,-179.475,8.756,149.550
C04415=1117.171,151.636,-61.609,-179.473,8.760,149.550
C04416=1117.166,151.884,-61.631,-179.471,8.764,149.551
C04417=1117.162,152.134,-61.653,-179.469,8.767,149.551
C04418=1117.157,152.382,-61.675,-179.466,8.770,149.551
C04419=1117.153,152.632,-61.697,-179.464,8.774,149.551
C04420=1117.147,152.881,-61.719,-179.462,8.777,149.551
C04421=1117.143,153.130,-61.741,-179.460,8.781,149.552
C04422=1117.139,153.378,-61.763,-179.457,8.784,149.552
C04423=1117.134,153.627,-61.785,-179.455,8.788,149.552
C04424=1117.130,153.877,-61.808,-179.452,8.792,149.552
C04425=1117.124,154.126,-61.830,-179.450,8.795,149.552
C04426=1117.120,154.375,-61.852,-179.448,8.798,149.552
C04427=1117.116,154.623,-61.874,-179.446,8.802,149.553
C04428=1117.111,154.872,-61.896,-179.443,8.805,149.553
C04429=1117.106,155.121,-61.919,-179.441,8.808,149.553
C04430=1117.102,155.370,-61.941,-179.439,8.812,149.553
C04431=1117.097,155.619,-61.963,-179.437,8.815,149.553
C04432=1117.092,155.868,-61.986,-179.434,8.819,149.553
C04433=1117.088,156.117,-62.008,-179.432,8.822,149.554
C04434=1117.083,156.366,-62.030,-179.430,8.825,149.554
C04435=1117.078,156.615,-62.053,-179.427,8.828,149.554
C04436=1117.074,156.864,-62.076,-179.425,8.832,149.554
C04437=1117.069,157.113,-62.097,-179.423,8.835,149.554
C04438=1117.065,157.327,-62.116,-179.421,8.838,149.554
C04439=1117.061,157.541,-62.136,-179.419,8.841,149.555
C04440=1117.057,157.755,-62.155,-179.417,8.844,149.555
C04441=1117.053,157.969,-62.174,-179.415,8.846,149.555
C04442=1117.049,158.182,-62.194,-179.413,8.849,149.555
C04443=1117.045,158.397,-62.213,-179.411,8.852,149.555
C04444=1117.041,158.609,-62.233,-179.409,8.855,149.555
C04445=1117.037,158.824,-62.252,-179.407,8.858,149.555
C04446=1117.033,159.072,-62.274,-179.405,8.862,149.555
C04447=1117.029,159.322,-62.296,-179.402,8.865,149.555
C04448=1117.023,159.570,-62.319,-179.401,8.867,149.556
C04449=1117.019,159.819,-62.342,-179.398,8.871,149.556
C04450=1117.014,160.068,-62.365,-179.396,8.874,149.556
C04451=1117.010,160.318,-62.387,-179.394,8.877,149.556
C04452=1117.005,160.566,-62.410,-179.392,8.881,149.556
C04453=1117.000,160.815,-62.432,-179.389,8.884,149.556
C04454=1116.997,161.064,-62.455,-179.387,8.887,149.556
C04455=1116.991,161.313,-62.477,-179.384,8.890,149.556
C04456=1116.987,161.562,-62.500,-179.382,8.893,149.556
C04457=1116.982,161.811,-62.523,-179.380,8.897,149.557
C04458=1116.978,162.060,-62.545,-179.377,8.900,149.557
C04459=1116.973,162.309,-62.568,-179.375,8.903,149.557
C04460=1116.969,162.557,-62.591,-179.373,8.906,149.557
C04461=1116.964,162.807,-62.614,-179.371,8.909,149.557
C04462=1116.960,163.056,-62.636,-179.369,8.912,149.557
C04463=1116.954,163.304,-62.659,-179.366,8.916,149.557
C04464=1116.949,163.554,-62.682,-179.364,8.919,149.558
C04465=1116.945,163.802,-62.705,-179.362,8.922,149.558
C04466=1116.941,164.051,-62.728,-179.360,8.926,149.558
C04467=1116.937,164.301,-62.750,-179.358,8.928,149.558
C04468=1116.931,164.549,-62.773,-179.355,8.931,149.558
C04469=1116.927,164.798,-62.796,-179.353,8.935,149.558
C04470=1116.923,165.047,-62.819,-179.351,8.938,149.558
C04471=1116.918,165.296,-62.843,-179.348,8.941,149.558
C04472=1116.914,165.545,-62.865,-179.346,8.944,149.558
C04473=1116.908,165.794,-62.888,-179.344,8.947,149.558
C04474=1116.904,166.042,-62.910,-179.342,8.950,149.559
C04475=1116.900,166.291,-62.934,-179.339,8.953,149.559
C04476=1116.895,166.540,-62.957,-179.337,8.956,149.559
C04477=1116.891,166.790,-62.979,-179.335,8.960,149.559
C04478=1116.885,167.038,-63.002,-179.333,8.962,149.559
C04479=1116.881,167.287,-63.026,-179.330,8.965,149.559
C04480=1116.877,167.536,-63.048,-179.328,8.969,149.559
C04481=1116.872,167.785,-63.072,-179.326,8.972,149.559
C04482=1116.867,168.034,-63.095,-179.323,8.975,149.559
C04483=1116.863,168.283,-63.118,-179.322,8.978,149.560
C04484=1116.859,168.532,-63.141,-179.319,8.981,149.560
C04485=1116.853,168.780,-63.164,-179.317,8.984,149.560
C04486=1116.849,169.029,-63.188,-179.315,8.987,149.560
C04487=1116.844,169.278,-63.211,-179.313,8.990,149.560
C04488=1116.840,169.527,-63.234,-179.310,8.993,149.560
C04489=1116.835,169.776,-63.257,-179.308,8.996,149.560
C04490=1116.831,170.025,-63.280,-179.306,8.999,149.560
C04491=1116.826,170.274,-63.304,-179.304,9.002,149.560
C04492=1116.822,170.522,-63.326,-179.301,9.005,149.560
C04493=1116.817,170.772,-63.350,-179.299,9.008,149.561
C04494=1116.813,170.985,-63.370,-179.297,9.011,149.561
C04495=1116.809,171.199,-63.390,-179.295,9.013,149.561
C04496=1116.805,171.413,-63.410,-179.294,9.016,149.561
C04497=1116.801,171.626,-63.430,-179.291,9.019,149.561
C04498=1116.797,171.840,-63.450,-179.289,9.021,149.561
C04499=1116.793,172.054,-63.470,-179.288,9.023,149.561
C04500=1116.789,172.267,-63.490,-179.286,9.026,149.561
C04501=1116.786,172.481,-63.509,-179.284,9.028,149.561
C04502=1116.781,172.730,-63.533,-179.282,9.032,149.561
C04503=1116.776,172.979,-63.556,-179.279,9.035,149.561
C04504=1116.771,173.228,-63.580,-179.278,9.037,149.562
C04505=1116.767,173.477,-63.603,-179.275,9.040,149.562
C04506=1116.762,173.725,-63.627,-179.273,9.044,149.562
C04507=1116.758,173.974,-63.650,-179.271,9.047,149.562
C04508=1116.753,174.223,-63.674,-179.269,9.049,149.562
C04509=1116.749,174.472,-63.696,-179.266,9.052,149.562
C04510=1116.744,174.721,-63.720,-179.264,9.056,149.562
C04511=1116.740,174.969,-63.744,-179.262,9.058,149.562
C04512=1116.735,175.218,-63.767,-179.260,9.061,149.562
C04513=1116.730,175.467,-63.791,-179.258,9.065,149.563
C04514=1116.726,175.716,-63.815,-179.256,9.067,149.563
C04515=1116.721,175.965,-63.838,-179.253,9.070,149.563
C04516=1116.717,176.214,-63.861,-179.251,9.073,149.563
C04517=1116.712,176.463,-63.885,-179.249,9.076,149.563
C04518=1116.708,176.711,-63.909,-179.247,9.079,149.563
C04519=1116.703,176.960,-63.932,-179.244,9.082,149.563
C04520=1116.698,177.209,-63.956,-179.243,9.085,149.563
C04521=1116.694,177.458,-63.980,-179.240,9.088,149.563
C04522=1116.690,177.708,-64.003,-179.238,9.091,149.563
C04523=1116.685,177.956,-64.027,-179.236,9.094,149.564
C04524=1116.681,178.205,-64.051,-179.234,9.097,149.564
C04525=1116.676,178.454,-64.074,-179.232,9.099,149.564
C04526=1116.672,178.702,-64.098,-179.230,9.103,149.564
C04527=1116.667,178.952,-64.122,-179.227,9.106,149.564
C04528=1116.662,179.200,-64.146,-179.225,9.108,149.564
C04529=1116.658,179.449,-64.169,-179.223,9.112,149.564
C04530=1116.653,179.697,-64.193,-179.221,9.115,149.564
C04531=1116.649,179.946,-64.216,-179.218,9.118,149.564
C04532=1116.644,180.195,-64.240,-179.215,9.122,149.564
C04533=1116.640,180.445,-64.264,-179.212,9.125,149.564
C04534=1116.636,180.693,-64.288,-179.210,9.128,149.564
C04535=1116.631,180.942,-64.312,-179.207,9.131,149.564
C04536=1116.626,181.191,-64.336,-179.204,9.134,149.564
C04537=1116.621,181.440,-64.360,-179.202,9.137,149.564
C04538=1116.617,181.688,-64.384,-179.199,9.140,149.564
C04539=1116.612,181.937,-64.408,-179.197,9.143,149.564
C04540=1116.608,182.186,-64.432,-179.194,9.146,149.564
C04541=1116.604,182.435,-64.456,-179.192,9.150,149.565
C04542=1116.599,182.684,-64.479,-179.189,9.153,149.565
C04543=1116.594,182.932,-64.504,-179.187,9.156,149.565
C04544=1116.590,183.181,-64.528,-179.184,9.159,149.565
C04545=1116.585,183.430,-64.551,-179.182,9.161,149.565
C04546=1116.581,183.679,-64.576,-179.180,9.164,149.565
C04547=1116.577,183.927,-64.600,-179.177,9.167,149.565
C04548=1116.571,184.177,-64.624,-179.174,9.170,149.565
C04549=1116.567,184.425,-64.648,-179.172,9.173,149.565
C04550=1116.564,184.638,-64.668,-179.170,9.176,149.565
C04551=1116.560,184.853,-64.689,-179.168,9.178,149.565
C04552=1116.555,185.066,-64.710,-179.166,9.181,149.565
C04553=1116.552,185.280,-64.730,-179.164,9.183,149.565
C04554=1116.548,185.494,-64.751,-179.162,9.186,149.565
C04555=1116.544,185.707,-64.772,-179.160,9.188,149.565
C04556=1116.540,185.920,-64.792,-179.157,9.191,149.565
C04557=1116.536,186.134,-64.814,-179.155,9.193,149.565
C04558=1116.532,186.383,-64.838,-179.153,9.197,149.565
C04559=1116.527,186.631,-64.862,-179.151,9.199,149.565
C04560=1116.522,186.880,-64.886,-179.148,9.202,149.565
C04561=1116.518,187.130,-64.910,-179.146,9.205,149.565
C04562=1116.513,187.378,-64.935,-179.144,9.207,149.565
C04563=1116.509,187.627,-64.959,-179.141,9.210,149.565
C04564=1116.504,187.875,-64.983,-179.139,9.213,149.565
C04565=1116.500,188.125,-65.008,-179.137,9.216,149.565
C04566=1116.496,188.373,-65.032,-179.134,9.219,149.565
C04567=1116.491,188.621,-65.056,-179.132,9.221,149.565
C04568=1116.486,188.870,-65.081,-179.130,9.224,149.565
C04569=1116.482,189.120,-65.105,-179.127,9.227,149.565
C04570=1116.477,189.369,-65.129,-179.125,9.230,149.565
C04571=1116.472,189.617,-65.153,-179.123,9.233,149.565
C04572=1116.469,189.866,-65.178,-179.121,9.235,149.565
C04573=1116.463,190.115,-65.202,-179.119,9.239,149.566
C04574=1116.459,190.363,-65.227,-179.117,9.241,149.566
C04575=1116.455,190.613,-65.252,-179.114,9.244,149.566
C04576=1116.450,190.861,-65.276,-179.113,9.246,149.566
C04577=1116.445,191.110,-65.300,-179.110,9.249,149.566
C04578=1116.442,191.358,-65.326,-179.108,9.252,149.566
C04579=1116.437,191.607,-65.350,-179.106,9.255,149.566
C04580=1116.432,191.855,-65.374,-179.104,9.257,149.566
C04581=1116.428,192.104,-65.399,-179.101,9.260,149.566
C04582=1116.423,192.353,-65.423,-179.099,9.263,149.566
C04583=1116.419,192.602,-65.447,-179.097,9.266,149.566
C04584=1116.414,192.851,-65.472,-179.095,9.268,149.566
C04585=1116.410,193.099,-65.497,-179.093,9.272,149.566
C04586=1116.405,193.348,-65.521,-179.091,9.274,149.566
C04587=1116.401,193.597,-65.546,-179.089,9.277,149.567
C04588=1116.396,193.845,-65.571,-179.087,9.280,149.567
C04589=1116.392,194.095,-65.595,-179.085,9.282,149.567
C04590=1116.387,194.343,-65.620,-179.082,9.285,149.567
C04591=1116.383,194.592,-65.644,-179.081,9.288,149.567
C04592=1116.378,194.841,-65.669,-179.079,9.290,149.567
C04593=1116.373,195.089,-65.695,-179.077,9.293,149.567
C04594=1116.370,195.338,-65.719,-179.075,9.296,149.567
C04595=1116.364,195.587,-65.744,-179.073,9.298,149.567
C04596=1116.360,195.835,-65.768,-179.071,9.302,149.568
C04597=1116.356,196.084,-65.794,-179.069,9.304,149.568
C04598=1116.351,196.333,-65.818,-179.068,9.307,149.568
C04599=1116.347,196.582,-65.843,-179.064,9.310,149.568
C04600=1116.342,196.831,-65.867,-179.062,9.313,149.568
C04601=1116.338,197.079,-65.893,-179.059,9.317,149.568
C04602=1116.333,197.328,-65.917,-179.056,9.320,149.568
C04603=1116.328,197.577,-65.942,-179.053,9.323,149.568
C04604=1116.324,197.825,-65.967,-179.049,9.327,149.568
C04605=1116.319,198.074,-65.992,-179.047,9.330,149.568
C04606=1116.316,198.288,-66.013,-179.044,9.333,149.568
C04607=1116.312,198.501,-66.034,-179.041,9.336,149.568
C04608=1116.308,198.714,-66.056,-179.040,9.338,149.568
C04609=1116.304,198.928,-66.078,-179.037,9.341,149.568
C04610=1116.300,199.142,-66.099,-179.034,9.344,149.568
C04611=1116.297,199.356,-66.121,-179.031,9.347,149.567
C04612=1116.293,199.569,-66.142,-179.029,9.349,149.567
C04613=1116.289,199.782,-66.164,-179.026,9.352,149.567
C04614=1116.284,200.031,-66.189,-179.023,9.354,149.567
C04615=1116.281,200.279,-66.214,-179.020,9.358,149.567
C04616=1116.276,200.528,-66.238,-179.017,9.361,149.567
C04617=1116.271,200.777,-66.264,-179.014,9.364,149.567
C04618=1116.266,201.026,-66.289,-179.012,9.367,149.567
C04619=1116.263,201.274,-66.314,-179.009,9.370,149.567
C04620=1116.258,201.523,-66.339,-179.005,9.373,149.567
C04621=1116.253,201.772,-66.364,-179.003,9.376,149.567
C04622=1116.249,202.021,-66.389,-179.000,9.379,149.567
C04623=1116.244,202.269,-66.415,-178.997,9.382,149.566
C04624=1116.241,202.518,-66.440,-178.994,9.384,149.566
C04625=1116.235,202.766,-66.465,-178.991,9.388,149.566
C04626=1116.231,203.015,-66.490,-178.988,9.391,149.566
C04627=1116.226,203.263,-66.516,-178.985,9.394,149.566
C04628=1116.222,203.513,-66.541,-178.982,9.397,149.566
C04629=1116.218,203.762,-66.567,-178.979,9.400,149.566
C04630=1116.213,204.009,-66.591,-178.976,9.402,149.566
C04631=1116.209,204.259,-66.616,-178.973,9.405,149.566
C04632=1116.204,204.507,-66.642,-178.970,9.408,149.566
C04633=1116.200,204.756,-66.667,-178.968,9.411,149.566
C04634=1116.196,205.005,-66.693,-178.965,9.414,149.565
C04635=1116.191,205.253,-66.719,-178.962,9.417,149.565
C04636=1116.186,205.502,-66.744,-178.959,9.419,149.565
C04637=1116.182,205.751,-66.769,-178.956,9.423,149.565
C04638=1116.177,205.999,-66.795,-178.953,9.426,149.565
C04639=1116.173,206.248,-66.821,-178.950,9.429,149.565
C04640=1116.169,206.497,-66.846,-178.947,9.432,149.565
C04641=1116.164,206.745,-66.871,-178.945,9.434,149.565
C04642=1116.159,206.994,-66.897,-178.942,9.437,149.565
C04643=1116.155,207.243,-66.922,-178.939,9.440,149.565
C04644=1116.150,207.491,-66.948,-178.936,9.443,149.565
C04645=1116.146,207.740,-66.974,-178.933,9.446,149.565
C04646=1116.142,207.989,-66.999,-178.931,9.449,149.565
C04647=1116.137,208.237,-67.025,-178.928,9.452,149.564
C04648=1116.133,208.486,-67.050,-178.925,9.454,149.564
C04649=1116.129,208.734,-67.076,-178.922,9.458,149.564
C04650=1116.124,208.983,-67.102,-178.919,9.460,149.564
C04651=1116.120,209.231,-67.127,-178.917,9.463,149.564
C04652=1116.115,209.480,-67.153,-178.914,9.466,149.564
C04653=1116.111,209.729,-67.179,-178.912,9.468,149.564
C04654=1116.106,209.977,-67.204,-178.909,9.471,149.564
C04655=1116.101,210.226,-67.231,-178.906,9.474,149.564
C04656=1116.097,210.475,-67.256,-178.903,9.477,149.564
C04657=1116.093,210.724,-67.282,-178.901,9.480,149.564
C04658=1116.088,210.972,-67.307,-178.898,9.483,149.564
C04659=1116.084,211.221,-67.333,-178.895,9.486,149.564
C04660=1116.080,211.469,-67.359,-178.893,9.489,149.564
C04661=1116.076,211.718,-67.385,-178.890,9.492,149.564
C04662=1116.071,211.932,-67.408,-178.887,9.495,149.564
C04663=1116.068,212.144,-67.429,-178.886,9.497,149.564
C04664=1116.063,212.358,-67.452,-178.884,9.500,149.564
C04665=1116.060,212.571,-67.474,-178.881,9.503,149.564
C04666=1116.057,212.785,-67.497,-178.879,9.505,149.564
C04667=1116.052,212.998,-67.519,-178.877,9.508,149.564
C04668=1116.049,213.212,-67.540,-178.875,9.511,149.564
C04669=1116.045,213.425,-67.563,-178.872,9.514,149.564
C04670=1116.041,213.674,-67.590,-178.870,9.516,149.564
C04671=1116.036,213.922,-67.615,-178.868,9.519,149.564
C04672=1116.032,214.170,-67.641,-178.866,9.521,149.564
C04673=1116.027,214.420,-67.667,-178.864,9.525,149.565
C04674=1116.023,214.668,-67.694,-178.862,9.527,149.565
C04675=1116.019,214.917,-67.719,-178.859,9.530,149.565
C04676=1116.014,215.165,-67.745,-178.858,9.533,149.565
C04677=1116.009,215.414,-67.771,-178.855,9.536,149.565
C04678=1116.005,215.663,-67.798,-178.853,9.539,149.565
C04679=1116.001,215.911,-67.823,-178.851,9.542,149.565
C04680=1115.997,216.159,-67.850,-178.849,9.545,149.565
C04681=1115.992,216.408,-67.876,-178.846,9.548,149.566
C04682=1115.987,216.657,-67.902,-178.845,9.551,149.566
C04683=1115.984,216.905,-67.928,-178.842,9.554,149.566
C04684=1115.979,217.154,-67.955,-178.840,9.557,149.566
C04685=1115.974,217.403,-67.980,-178.838,9.559,149.566
C04686=1115.970,217.651,-68.007,-178.835,9.563,149.566
C04687=1115.965,217.900,-68.033,-178.833,9.566,149.566
C04688=1115.962,218.148,-68.060,-178.831,9.569,149.566
C04689=1115.957,218.397,-68.085,-178.829,9.571,149.566
C04690=1115.952,218.645,-68.112,-178.826,9.575,149.566
C04691=1115.948,218.894,-68.138,-178.824,9.578,149.567
C04692=1115.944,219.142,-68.164,-178.822,9.581,149.567
C04693=1115.939,219.391,-68.191,-178.819,9.584,149.567
C04694=1115.935,219.639,-68.217,-178.817,9.587,149.567
C04695=1115.930,219.888,-68.244,-178.814,9.590,149.567
C04696=1115.926,220.137,-68.270,-178.812,9.593,149.567
C04697=1115.921,220.386,-68.296,-178.810,9.596,149.567
C04698=1115.917,220.634,-68.323,-178.808,9.599,149.567
C04699=1115.913,220.883,-68.349,-178.805,9.603,149.567
C04700=1115.908,221.131,-68.376,-178.803,9.606,149.568
C04701=1115.904,221.379,-68.402,-178.800,9.609,149.568
C04702=1115.900,221.629,-68.428,-178.798,9.612,149.568
C04703=1115.896,221.877,-68.455,-178.795,9.615,149.568
C04704=1115.891,222.125,-68.482,-178.793,9.618,149.568
C04705=1115.887,222.374,-68.508,-178.790,9.621,149.568
C04706=1115.882,222.623,-68.535,-178.787,9.624,149.568
C04707=1115.878,222.871,-68.561,-178.785,9.627,149.568
C04708=1115.873,223.120,-68.588,-178.782,9.631,149.568
C04709=1115.869,223.368,-68.614,-178.780,9.634,149.568
C04710=1115.865,223.616,-68.641,-178.777,9.637,149.568
C04711=1115.860,223.866,-68.667,-178.775,9.640,149.568
C04712=1115.856,224.114,-68.694,-178.772,9.643,149.568
C04713=1115.851,224.362,-68.721,-178.770,9.646,149.568
C04714=1115.847,224.610,-68.747,-178.767,9.650,149.568
C04715=1115.842,224.860,-68.774,-178.764,9.653,149.568
C04716=1115.838,225.108,-68.800,-178.761,9.656,149.568
C04717=1115.834,225.356,-68.827,-178.759,9.659,149.568
C04718=1115.830,225.569,-68.851,-178.757,9.661,149.569
C04719=1115.826,225.783,-68.874,-178.754,9.664,149.569
C04720=1115.823,225.996,-68.896,-178.751,9.667,149.568
C04721=1115.819,226.209,-68.919,-178.749,9.669,149.569
C04722=1115.815,226.423,-68.942,-178.747,9.673,149.569
C04723=1115.811,226.636,-68.966,-178.745,9.675,149.568
C04724=1115.807,226.850,-68.988,-178.742,9.678,149.569
C04725=1115.804,227.062,-69.011,-178.739,9.681,149.569
C04726=1115.799,227.311,-69.038,-178.737,9.683,149.568
C04727=1115.795,227.559,-69.065,-178.734,9.687,149.569
C04728=1115.791,227.807,-69.092,-178.731,9.689,149.568
C04729=1115.786,228.056,-69.119,-178.729,9.692,149.568
C04730=1115.782,228.305,-69.146,-178.725,9.696,149.568
C04731=1115.778,228.553,-69.173,-178.722,9.699,149.568
C04732=1115.773,228.802,-69.200,-178.719,9.702,149.568
C04733=1115.769,229.050,-69.227,-178.717,9.705,149.568
C04734=1115.764,229.299,-69.254,-178.713,9.708,149.568
C04735=1115.760,229.547,-69.281,-178.710,9.711,149.568
C04736=1115.756,229.796,-69.308,-178.708,9.714,149.568
C04737=1115.752,230.045,-69.335,-178.704,9.718,149.568
C04738=1115.747,230.293,-69.362,-178.701,9.721,149.568
C04739=1115.742,230.542,-69.389,-178.698,9.723,149.568
C04740=1115.738,230.790,-69.416,-178.696,9.726,149.568
C04741=1115.734,231.038,-69.443,-178.692,9.730,149.568
C04742=1115.730,231.287,-69.471,-178.689,9.733,149.568
C04743=1115.725,231.535,-69.498,-178.686,9.735,149.568
C04744=1115.721,231.784,-69.525,-178.684,9.738,149.567
C04745=1115.716,232.032,-69.552,-178.681,9.741,149.567
C04746=1115.712,232.281,-69.578,-178.678,9.744,149.567
C04747=1115.708,232.529,-69.607,-178.675,9.747,149.567
C04748=1115.704,232.778,-69.634,-178.672,9.750,149.567
C04749=1115.699,233.026,-69.661,-178.669,9.752,149.567
C04750=1115.694,233.275,-69.688,-178.666,9.755,149.567
C04751=1115.691,233.523,-69.716,-178.664,9.758,149.567
C04752=1115.686,233.772,-69.743,-178.661,9.761,149.567
C04753=1115.681,234.020,-69.770,-178.658,9.764,149.567
C04754=1115.677,234.268,-69.798,-178.655,9.766,149.567
C04755=1115.673,234.517,-69.825,-178.652,9.769,149.566
C04756=1115.669,234.766,-69.852,-178.649,9.772,149.566
C04757=1115.665,235.013,-69.880,-178.646,9.775,149.566
C04758=1115.661,235.263,-69.907,-178.644,9.777,149.566
C04759=1115.656,235.511,-69.934,-178.641,9.780,149.566
C04760=1115.651,235.759,-69.962,-178.638,9.782,149.566
C04761=1115.647,236.008,-69.989,-178.635,9.785,149.566
C04762=1115.643,236.256,-70.017,-178.632,9.788,149.566
C04763=1115.638,236.505,-70.044,-178.630,9.790,149.566
C04764=1115.634,236.752,-70.072,-178.628,9.793,149.566
C04765=1115.630,237.002,-70.099,-178.625,9.796,149.566
C04766=1115.626,237.249,-70.127,-178.622,9.799,149.565
C04767=1115.621,237.498,-70.154,-178.619,9.801,149.565
C04768=1115.617,237.747,-70.183,-178.616,9.803,149.565
C04769=1115.612,237.995,-70.210,-178.614,9.806,149.565
C04770=1115.608,238.244,-70.238,-178.612,9.808,149.565
C04771=1115.603,238.492,-70.265,-178.609,9.811,149.565
C04772=1115.599,238.740,-70.293,-178.606,9.814,149.565
C04773=1115.595,238.990,-70.320,-178.604,9.816,149.565
C04774=1115.591,239.203,-70.344,-178.601,9.818,149.565
C04775=1115.588,239.416,-70.367,-178.599,9.820,149.565
C04776=1115.584,239.628,-70.392,-178.597,9.823,149.565
C04777=1115.580,239.841,-70.416,-178.594,9.825,149.565
C04778=1115.577,240.055,-70.439,-178.592,9.828,149.565
C04779=1115.573,240.268,-70.463,-178.590,9.830,149.564
C04780=1115.569,240.481,-70.486,-178.588,9.832,149.565
C04781=1115.565,240.694,-70.510,-178.586,9.834,149.564
C04782=1115.561,240.943,-70.539,-178.584,9.836,149.564
C04783=1115.557,241.191,-70.567,-178.581,9.839,149.564
C04784=1115.552,241.439,-70.594,-178.579,9.841,149.564
C04785=1115.548,241.688,-70.622,-178.576,9.844,149.564
C04786=1115.544,241.936,-70.649,-178.574,9.846,149.564
C04787=1115.540,242.185,-70.677,-178.571,9.849,149.564
C04788=1115.535,242.433,-70.705,-178.569,9.851,149.564
C04789=1115.531,242.682,-70.733,-178.567,9.854,149.564
C04790=1115.527,242.930,-70.761,-178.564,9.856,149.564
C04791=1115.522,243.178,-70.788,-178.562,9.859,149.564
C04792=1115.518,243.427,-70.816,-178.560,9.862,149.564
C04793=1115.513,243.675,-70.845,-178.557,9.864,149.564
C04794=1115.509,243.923,-70.873,-178.555,9.867,149.564
C04795=1115.505,244.171,-70.901,-178.553,9.869,149.564
C04796=1115.501,244.420,-70.929,-178.551,9.871,149.564
C04797=1115.496,244.669,-70.957,-178.548,9.874,149.564
C04798=1115.492,244.917,-70.985,-178.546,9.876,149.564
C04799=1115.488,245.165,-71.012,-178.544,9.879,149.564
C04800=1115.483,245.414,-71.041,-178.542,9.882,149.564
C04801=1115.479,245.662,-71.069,-178.540,9.884,149.564
C04802=1115.475,245.911,-71.097,-178.538,9.886,149.564
C04803=1115.471,246.158,-71.125,-178.535,9.889,149.564
C04804=1115.466,246.407,-71.154,-178.533,9.892,149.564
C04805=1115.462,246.656,-71.181,-178.531,9.894,149.564
C04806=1115.458,246.904,-71.209,-178.529,9.897,149.565
C04807=1115.453,247.153,-71.237,-178.527,9.899,149.565
C04808=1115.449,247.401,-71.265,-178.525,9.902,149.565
C04809=1115.445,247.649,-71.293,-178.522,9.906,149.565
C04810=1115.440,247.898,-71.322,-178.517,9.910,149.564
C04811=1115.436,248.146,-71.350,-178.513,9.913,149.564
C04812=1115.431,248.395,-71.378,-178.509,9.917,149.564
C04813=1115.427,248.643,-71.406,-178.505,9.920,149.564
C04814=1115.423,248.891,-71.434,-178.500,9.924,149.564
C04815=1115.419,249.139,-71.464,-178.497,9.928,149.563
C04816=1115.415,249.387,-71.491,-178.493,9.931,149.563
C04817=1115.410,249.636,-71.520,-178.489,9.934,149.563
C04818=1115.406,249.884,-71.548,-178.485,9.937,149.563
C04819=1115.401,250.133,-71.577,-178.482,9.940,149.562
C04820=1115.398,250.381,-71.605,-178.478,9.943,149.562
C04821=1115.393,250.630,-71.633,-178.475,9.946,149.562
C04822=1115.389,250.878,-71.662,-178.471,9.949,149.562
C04823=1115.384,251.126,-71.690,-178.468,9.952,149.561
C04824=1115.380,251.374,-71.719,-178.465,9.954,149.561
C04825=1115.376,251.623,-71.747,-178.462,9.957,149.561
C04826=1115.372,251.871,-71.776,-178.458,9.959,149.561
C04827=1115.367,252.119,-71.805,-178.456,9.962,149.561
C04828=1115.363,252.368,-71.833,-178.453,9.964,149.561
C04829=1115.358,252.616,-71.861,-178.450,9.967,149.560
C04830=1115.356,252.829,-71.886,-178.448,9.969,149.560
C04831=1115.351,253.042,-71.911,-178.446,9.971,149.560
C04832=1115.349,253.255,-71.935,-178.443,9.973,149.560
C04833=1115.344,253.468,-71.960,-178.441,9.975,149.560
C04834=1115.340,253.681,-71.984,-178.439,9.976,149.560
C04835=1115.337,253.894,-72.009,-178.437,9.978,149.560
C04836=1115.333,254.107,-72.033,-178.435,9.980,149.560
C04837=1115.330,254.320,-72.058,-178.434,9.982,149.560
C04838=1115.325,254.568,-72.086,-178.432,9.984,149.560
C04839=1115.321,254.816,-72.116,-178.430,9.986,149.560
C04840=1115.317,255.065,-72.144,-178.428,9.988,149.560
C04841=1115.313,255.314,-72.173,-178.427,9.990,149.560
C04842=1115.308,255.562,-72.202,-178.425,9.992,149.560
C04843=1115.304,255.810,-72.230,-178.423,9.994,149.560
C04844=1115.300,256.058,-72.259,-178.422,9.996,149.560
C04845=1115.295,256.307,-72.288,-178.419,9.998,149.560
C04846=1115.291,256.555,-72.317,-178.416,10.001,149.560
C04847=1115.287,256.803,-72.345,-178.414,10.004,149.560
C04848=1115.283,257.052,-72.375,-178.411,10.007,149.560
C04849=1115.278,257.300,-72.403,-178.408,10.010,149.560
C04850=1115.274,257.548,-72.432,-178.405,10.012,149.560
C04851=1115.270,257.797,-72.461,-178.402,10.016,149.560
C04852=1115.266,258.045,-72.490,-178.399,10.018,149.560
C04853=1115.261,258.293,-72.518,-178.396,10.021,149.559
C04854=1115.257,258.541,-72.547,-178.394,10.024,149.559
C04855=1115.252,258.790,-72.576,-178.391,10.027,149.559
C04856=1115.249,259.038,-72.605,-178.388,10.029,149.559
C04857=1115.244,259.286,-72.634,-178.385,10.032,149.559
C04858=1115.240,259.534,-72.663,-178.382,10.035,149.559
C04859=1115.236,259.783,-72.692,-178.379,10.038,149.559
C04860=1115.232,260.031,-72.721,-178.376,10.041,149.559
C04861=1115.228,260.280,-72.750,-178.373,10.043,149.559
C04862=1115.223,260.527,-72.779,-178.370,10.046,149.559
C04863=1115.219,260.775,-72.808,-178.367,10.049,149.559
C04864=1115.214,261.024,-72.837,-178.365,10.052,149.558
C04865=1115.211,261.272,-72.866,-178.362,10.054,149.558
C04866=1115.207,261.520,-72.896,-178.358,10.057,149.558
C04867=1115.202,261.769,-72.925,-178.355,10.060,149.558
C04868=1115.197,262.017,-72.953,-178.352,10.063,149.558
C04869=1115.193,262.265,-72.983,-178.349,10.066,149.558
C04870=1115.189,262.513,-73.012,-178.346,10.069,149.558
C04871=1115.185,262.762,-73.042,-178.343,10.071,149.558
C04872=1115.181,263.010,-73.071,-178.340,10.074,149.557
C04873=1115.176,263.259,-73.100,-178.337,10.077,149.557
C04874=1115.173,263.507,-73.129,-178.334,10.079,149.557
C04875=1115.168,263.755,-73.158,-178.330,10.083,149.557
C04876=1115.164,264.003,-73.187,-178.327,10.085,149.557
C04877=1115.160,264.251,-73.217,-178.324,10.088,149.557
C04878=1115.155,264.499,-73.246,-178.320,10.090,149.556
C04879=1115.151,264.747,-73.276,-178.318,10.093,149.556
C04880=1115.147,264.996,-73.305,-178.315,10.095,149.556
C04881=1115.143,265.244,-73.335,-178.312,10.098,149.556
C04882=1115.139,265.492,-73.364,-178.309,10.101,149.556
C04883=1115.134,265.741,-73.393,-178.307,10.103,149.556
C04884=1115.130,265.989,-73.423,-178.304,10.105,149.556
C04885=1115.126,266.237,-73.452,-178.301,10.108,149.555
C04886=1115.122,266.450,-73.477,-178.299,10.110,149.555
C04887=1115.118,266.663,-73.502,-178.297,10.112,149.555
C04888=1115.114,266.875,-73.528,-178.295,10.115,149.555
C04889=1115.111,267.089,-73.553,-178.292,10.117,149.555
C04890=1115.108,267.301,-73.579,-178.290,10.118,149.555
C04891=1115.103,267.514,-73.604,-178.287,10.121,149.555
C04892=1115.100,267.728,-73.629,-178.285,10.123,149.555
C04893=1115.097,267.940,-73.655,-178.282,10.125,149.555
C04894=1115.092,268.189,-73.684,-178.280,10.128,149.555
C04895=1115.088,268.437,-73.714,-178.277,10.130,149.554
C04896=1115.084,268.685,-73.743,-178.274,10.133,149.554
C04897=1115.080,268.933,-73.773,-178.271,10.135,149.554
C04898=1115.076,269.181,-73.803,-178.268,10.138,149.554
C04899=1115.071,269.430,-73.833,-178.266,10.140,149.554
C04900=1115.067,269.678,-73.862,-178.263,10.143,149.554
C04901=1115.063,269.926,-73.892,-178.260,10.146,149.554
C04902=1115.059,270.175,-73.921,-178.257,10.148,149.554
C04903=1115.055,270.422,-73.951,-178.254,10.151,149.554
C04904=1115.051,270.670,-73.981,-178.252,10.153,149.554
C04905=1115.046,270.919,-74.010,-178.249,10.156,149.553
C04906=1115.041,271.167,-74.040,-178.246,10.159,149.553
C04907=1115.038,271.415,-74.071,-178.243,10.162,149.553
C04908=1115.033,271.663,-74.100,-178.240,10.164,149.553
C04909=1115.029,271.911,-74.129,-178.237,10.167,149.553
C04910=1115.025,272.159,-74.160,-178.235,10.169,149.553
C04911=1115.020,272.408,-74.190,-178.232,10.172,149.553
C04912=1115.016,272.656,-74.219,-178.229,10.175,149.553
C04913=1115.012,272.904,-74.249,-178.226,10.177,149.552
C04914=1115.008,273.152,-74.279,-178.223,10.180,149.552
C04915=1115.003,273.400,-74.309,-178.220,10.182,149.552
C04916=1114.999,273.648,-74.339,-178.217,10.185,149.552
C04917=1114.996,273.897,-74.369,-178.215,10.187,149.552
C04918=1114.992,274.145,-74.399,-178.212,10.190,149.552
C04919=1114.987,274.393,-74.429,-178.209,10.193,149.552
C04920=1114.983,274.642,-74.458,-178.206,10.196,149.552
C04921=1114.979,274.889,-74.489,-178.203,10.198,149.552
C04922=1114.974,275.138,-74.519,-178.200,10.201,149.551
C04923=1114.970,275.385,-74.549,-178.197,10.203,149.551
C04924=1114.966,275.634,-74.578,-178.194,10.206,149.551
C04925=1114.962,275.882,-74.609,-178.191,10.209,149.551
C04926=1114.958,276.130,-74.640,-178.188,10.212,149.551
C04927=1114.954,276.378,-74.669,-178.185,10.214,149.551
C04928=1114.949,276.626,-74.700,-178.182,10.217,149.551
C04929=1114.945,276.874,-74.729,-178.179,10.220,149.550
C04930=1114.941,277.122,-74.759,-178.176,10.222,149.550
C04931=1114.937,277.371,-74.790,-178.172,10.225,149.550
C04932=1114.933,277.619,-74.820,-178.169,10.228,149.550
C04933=1114.929,277.867,-74.850,-178.167,10.230,149.550
C04934=1114.924,278.115,-74.880,-178.164,10.233,149.550
C04935=1114.920,278.363,-74.910,-178.160,10.236,149.550
C04936=1114.916,278.612,-74.942,-178.157,10.238,149.549
C04937=1114.912,278.860,-74.971,-178.154,10.241,149.549
C04938=1114.908,279.108,-75.002,-178.151,10.243,149.549
C04939=1114.904,279.355,-75.032,-178.148,10.246,149.549
C04940=1114.899,279.603,-75.063,-178.145,10.249,149.549
C04941=1114.895,279.852,-75.093,-178.142,10.251,149.549
C04942=1114.892,280.065,-75.118,-178.139,10.253,149.548
C04943=1114.888,280.278,-75.145,-178.137,10.256,149.548
C04944=1114.884,280.490,-75.170,-178.134,10.258,149.548
C04945=1114.881,280.703,-75.197,-178.132,10.260,149.548
C04946=1114.877,280.916,-75.224,-178.129,10.263,149.548
C04947=1114.874,281.128,-75.249,-178.126,10.265,149.548
C04948=1114.870,281.342,-75.276,-178.123,10.267,149.547
C04949=1114.866,281.554,-75.301,-178.121,10.269,149.547
C04950=1114.863,281.802,-75.332,-178.118,10.272,149.547
C04951=1114.858,282.050,-75.363,-178.114,10.274,149.547
C04952=1114.854,282.298,-75.394,-178.111,10.277,149.547
C04953=1114.850,282.547,-75.423,-178.108,10.279,149.547
C04954=1114.846,282.795,-75.454,-178.105,10.282,149.546
C04955=1114.842,283.042,-75.484,-178.102,10.285,149.546
C04956=1114.837,283.290,-75.515,-178.099,10.287,149.546
C04957=1114.833,283.539,-75.546,-178.097,10.289,149.546
C04958=1114.829,283.787,-75.576,-178.093,10.292,149.546
C04959=1114.825,284.035,-75.607,-178.090,10.294,149.546
C04960=1114.821,284.283,-75.638,-178.087,10.297,149.546
C04961=1114.817,284.531,-75.668,-178.084,10.300,149.545
C04962=1114.812,284.779,-75.699,-178.081,10.302,149.545
C04963=1114.808,285.028,-75.730,-178.078,10.305,149.545
C04964=1114.804,285.275,-75.760,-178.075,10.308,149.545
C04965=1114.800,285.523,-75.791,-178.072,10.309,149.544
C04966=1114.796,285.772,-75.822,-178.069,10.312,149.544
C04967=1114.792,286.019,-75.853,-178.066,10.315,149.544
C04968=1114.787,286.267,-75.884,-178.063,10.317,149.544
C04969=1114.783,286.516,-75.915,-178.060,10.320,149.544
C04970=1114.779,286.763,-75.946,-178.057,10.322,149.544
C04971=1114.776,287.012,-75.976,-178.054,10.325,149.544
C04972=1114.771,287.260,-76.007,-178.050,10.328,149.543
C04973=1114.766,287.508,-76.038,-178.047,10.330,149.543
C04974=1114.763,287.756,-76.070,-178.045,10.332,149.543
C04975=1114.759,288.003,-76.100,-178.042,10.335,149.543
C04976=1114.755,288.252,-76.131,-178.039,10.337,149.543
C04977=1114.750,288.500,-76.162,-178.035,10.340,149.542
C04978=1114.746,288.747,-76.193,-178.033,10.343,149.542
C04979=1114.743,288.996,-76.224,-178.029,10.345,149.542
C04980=1114.738,289.244,-76.255,-178.026,10.348,149.542
C04981=1114.734,289.492,-76.286,-178.023,10.350,149.542
C04982=1114.730,289.740,-76.317,-178.020,10.353,149.542
C04983=1114.726,289.988,-76.348,-178.018,10.355,149.542
C04984=1114.721,290.236,-76.379,-178.014,10.357,149.541
C04985=1114.717,290.484,-76.411,-178.011,10.360,149.541
C04986=1114.713,290.732,-76.441,-178.008,10.363,149.541
C04987=1114.709,290.981,-76.472,-178.005,10.365,149.541
C04988=1114.705,291.228,-76.504,-178.002,10.368,149.541
C04989=1114.701,291.477,-76.535,-177.999,10.371,149.540
C04990=1114.697,291.724,-76.566,-177.996,10.373,149.540
C04991=1114.693,291.973,-76.598,-177.993,10.376,149.540
C04992=1114.688,292.220,-76.629,-177.990,10.378,149.540
C04993=1114.684,292.469,-76.660,-177.987,10.380,149.540
C04994=1114.680,292.717,-76.691,-177.984,10.383,149.540
C04995=1114.676,292.965,-76.723,-177.981,10.385,149.539
C04996=1114.672,293.212,-76.753,-177.978,10.388,149.539
C04997=1114.669,293.460,-76.785,-177.974,10.391,149.539
C04998=1114.665,293.673,-76.812,-177.972,10.393,149.539
C04999=1114.661,293.886,-76.838,-177.969,10.395,149.539
C05000=1114.657,294.098,-76.866,-177.966,10.397,149.538
C05001=1114.654,294.311,-76.892,-177.964,10.399,149.538
C05002=1114.651,294.523,-76.919,-177.961,10.402,149.538
C05003=1114.647,294.736,-76.946,-177.959,10.404,149.538
C05004=1114.644,294.948,-76.973,-177.956,10.405,149.538
C05005=1114.640,295.161,-77.000,-177.953,10.408,149.538
C05006=1114.636,295.409,-77.032,-177.950,10.411,149.538
C05007=1114.632,295.657,-77.062,-177.948,10.413,149.537
C05008=1114.628,295.905,-77.094,-177.945,10.415,149.537
C05009=1114.624,296.153,-77.126,-177.941,10.418,149.537
C05010=1114.620,296.401,-77.157,-177.938,10.421,149.537
C05011=1114.615,296.649,-77.189,-177.935,10.423,149.537
C05012=1114.611,296.897,-77.221,-177.932,10.426,149.537
C05013=1114.607,297.145,-77.252,-177.929,10.428,149.536
C05014=1114.603,297.393,-77.284,-177.926,10.431,149.536
C05015=1114.599,297.641,-77.315,-177.923,10.433,149.536
C05016=1114.595,297.889,-77.347,-177.920,10.435,149.536
C05017=1114.590,298.137,-77.378,-177.917,10.438,149.536
C05018=1114.587,298.385,-77.410,-177.914,10.441,149.536
C05019=1114.582,298.633,-77.442,-177.911,10.443,149.535
C05020=1114.578,298.880,-77.474,-177.908,10.446,149.535
C05021=1114.574,299.128,-77.505,-177.904,10.448,149.535
C05022=1114.570,299.377,-77.537,-177.902,10.451,149.535
C05023=1114.566,299.624,-77.568,-177.898,10.453,149.535
C05024=1114.562,299.872,-77.600,-177.895,10.456,149.535
C05025=1114.558,300.121,-77.632,-177.892,10.459,149.534
C05026=1114.553,300.368,-77.664,-177.890,10.461,149.534
C05027=1114.550,300.616,-77.696,-177.886,10.463,149.534
C05028=1114.546,300.864,-77.728,-177.883,10.466,149.534
C05029=1114.541,301.112,-77.760,-177.880,10.468,149.534
C05030=1114.537,301.360,-77.791,-177.877,10.471,149.533
C05031=1114.534,301.608,-77.823,-177.874,10.473,149.533
C05032=1114.529,301.855,-77.855,-177.871,10.476,149.533
C05033=1114.525,302.104,-77.887,-177.867,10.479,149.533
C05034=1114.521,302.352,-77.919,-177.865,10.481,149.533
C05035=1114.517,302.600,-77.951,-177.861,10.484,149.533
C05036=1114.512,302.847,-77.983,-177.859,10.486,149.532
C05037=1114.509,303.095,-78.015,-177.856,10.488,149.532
C05038=1114.505,303.343,-78.047,-177.853,10.491,149.532
C05039=1114.500,303.591,-78.079,-177.849,10.493,149.532
C05040=1114.496,303.839,-78.111,-177.846,10.496,149.532
C05041=1114.493,304.087,-78.142,-177.843,10.499,149.531
C05042=1114.488,304.335,-78.175,-177.840,10.501,149.531
C05043=1114.484,304.583,-78.206,-177.837,10.504,149.531
C05044=1114.480,304.830,-78.239,-177.834,10.507,149.531
C05045=1114.476,305.079,-78.271,-177.831,10.509,149.531
C05046=1114.472,305.327,-78.303,-177.828,10.511,149.531
C05047=1114.467,305.574,-78.335,-177.825,10.513,149.530
C05048=1114.463,305.822,-78.367,-177.822,10.516,149.530
C05049=1114.459,306.070,-78.400,-177.819,10.519,149.530
C05050=1114.456,306.318,-78.432,-177.816,10.521,149.530
C05051=1114.452,306.566,-78.464,-177.812,10.524,149.530
C05052=1114.447,306.814,-78.496,-177.809,10.526,149.529
C05053=1114.443,307.061,-78.529,-177.806,10.529,149.529
C05054=1114.440,307.274,-78.556,-177.804,10.531,149.529
C05055=1114.436,307.487,-78.584,-177.801,10.533,149.529
C05056=1114.433,307.699,-78.612,-177.798,10.535,149.529
C05057=1114.429,307.911,-78.639,-177.796,10.537,149.529
C05058=1114.426,308.124,-78.667,-177.793,10.539,149.529
C05059=1114.422,308.336,-78.695,-177.790,10.542,149.528
C05060=1114.419,308.548,-78.723,-177.788,10.544,149.528
C05061=1114.416,308.762,-78.750,-177.785,10.546,149.528
C05062=1114.411,309.009,-78.782,-177.782,10.548,149.528
C05063=1114.408,309.257,-78.815,-177.779,10.551,149.528
C05064=1114.403,309.505,-78.847,-177.776,10.554,149.528
C05065=1114.399,309.753,-78.880,-177.773,10.556,149.527
C05066=1114.395,310.001,-78.912,-177.770,10.559,149.527
C05067=1114.391,310.248,-78.945,-177.767,10.561,149.527
C05068=1114.387,310.496,-78.977,-177.763,10.564,149.527
C05069=1114.383,310.744,-79.010,-177.760,10.566,149.527
C05070=1114.379,310.992,-79.042,-177.757,10.569,149.526
C05071=1114.375,311.239,-79.075,-177.754,10.572,149.526
C05072=1114.370,311.488,-79.107,-177.751,10.573,149.526
C05073=1114.367,311.735,-79.140,-177.748,10.576,149.526
C05074=1114.363,311.983,-79.172,-177.745,10.578,149.526
C05075=1114.359,312.231,-79.205,-177.742,10.581,149.526
C05076=1114.355,312.479,-79.237,-177.739,10.584,149.525
C05077=1114.351,312.727,-79.271,-177.735,10.586,149.525
C05078=1114.347,312.974,-79.303,-177.733,10.589,149.525
C05079=1114.343,313.223,-79.336,-177.729,10.591,149.525
C05080=1114.339,313.470,-79.369,-177.726,10.594,149.525
C05081=1114.335,313.718,-79.401,-177.723,10.597,149.525
C05082=1114.331,313.966,-79.434,-177.720,10.598,149.524
C05083=1114.327,314.214,-79.467,-177.717,10.601,149.524
C05084=1114.322,314.462,-79.500,-177.714,10.603,149.524
C05085=1114.319,314.710,-79.532,-177.711,10.606,149.524
C05086=1114.315,314.957,-79.565,-177.708,10.609,149.524
C05087=1114.310,315.205,-79.598,-177.705,10.611,149.524
C05088=1114.307,315.453,-79.631,-177.702,10.614,149.523
C05089=1114.303,315.701,-79.663,-177.698,10.616,149.523
C05090=1114.298,315.949,-79.696,-177.695,10.619,149.523
C05091=1114.294,316.196,-79.729,-177.692,10.621,149.523
C05092=1114.291,316.444,-79.762,-177.689,10.624,149.523
C05093=1114.287,316.691,-79.795,-177.686,10.626,149.522
C05094=1114.282,316.940,-79.828,-177.683,10.628,149.522
C05095=1114.278,317.188,-79.861,-177.680,10.631,149.522
C05096=1114.274,317.435,-79.894,-177.677,10.634,149.522
C05097=1114.271,317.683,-79.927,-177.674,10.636,149.522
C05098=1114.267,317.930,-79.960,-177.670,10.639,149.522
C05099=1114.262,318.178,-79.993,-177.667,10.641,149.521
C05100=1114.258,318.426,-80.026,-177.664,10.644,149.521
C05101=1114.254,318.674,-80.059,-177.661,10.646,149.521
C05102=1114.250,318.921,-80.092,-177.658,10.649,149.521
C05103=1114.247,319.169,-80.125,-177.655,10.652,149.521
C05104=1114.243,319.417,-80.158,-177.652,10.653,149.520
C05105=1114.239,319.665,-80.192,-177.649,10.656,149.520
C05106=1114.235,319.913,-80.225,-177.646,10.659,149.520
C05107=1114.231,320.160,-80.258,-177.642,10.661,149.520
C05108=1114.226,320.408,-80.291,-177.639,10.664,149.520
C05109=1114.222,320.656,-80.324,-177.636,10.666,149.519
C05110=1114.220,320.868,-80.352,-177.634,10.668,149.519
C05111=1114.215,321.081,-80.381,-177.631,10.671,149.519
C05112=1114.213,321.293,-80.409,-177.628,10.673,149.519
C05113=1114.209,321.505,-80.438,-177.626,10.675,149.519
C05114=1114.206,321.718,-80.466,-177.623,10.677,149.519
C05115=1114.202,321.930,-80.495,-177.620,10.679,149.519
C05116=1114.199,322.142,-80.524,-177.618,10.681,149.518
C05117=1114.195,322.354,-80.552,-177.615,10.684,149.518
C05118=1114.192,322.603,-80.586,-177.611,10.686,149.518
C05119=1114.187,322.850,-80.619,-177.608,10.689,149.518
C05120=1114.183,323.098,-80.652,-177.606,10.690,149.518
C05121=1114.179,323.346,-80.685,-177.602,10.693,149.517
C05122=1114.175,323.593,-80.719,-177.600,10.696,149.517
C05123=1114.171,323.841,-80.752,-177.596,10.698,149.517
C05124=1114.168,324.089,-80.786,-177.593,10.701,149.517
C05125=1114.163,324.337,-80.819,-177.590,10.703,149.517
C05126=1114.160,324.584,-80.853,-177.587,10.706,149.517
C05127=1114.155,324.832,-80.886,-177.584,10.709,149.516
C05128=1114.151,325.079,-80.919,-177.580,10.711,149.516
C05129=1114.148,325.327,-80.953,-177.577,10.713,149.516
C05130=1114.144,325.575,-80.986,-177.574,10.716,149.516
C05131=1114.140,325.823,-81.020,-177.571,10.718,149.516
C05132=1114.135,326.070,-81.054,-177.568,10.720,149.515
C05133=1114.132,326.318,-81.088,-177.565,10.723,149.515
C05134=1114.128,326.566,-81.121,-177.562,10.726,149.515
C05135=1114.124,326.813,-81.155,-177.559,10.728,149.515
C05136=1114.120,327.061,-81.188,-177.556,10.731,149.515
C05137=1114.116,327.309,-81.222,-177.552,10.733,149.515
C05138=1114.112,327.557,-81.256,-177.549,10.736,149.514
C05139=1114.108,327.804,-81.290,-177.546,10.738,149.514
C05140=1114.104,328.052,-81.323,-177.543,10.741,149.514
C05141=1114.100,328.300,-81.357,-177.539,10.743,149.514
C05142=1114.096,328.547,-81.390,-177.537,10.745,149.514
C05143=1114.092,328.795,-81.425,-177.534,10.748,149.513
C05144=1114.088,329.043,-81.458,-177.530,10.750,149.513
C05145=1114.084,329.290,-81.492,-177.527,10.753,149.513
C05146=1114.080,329.538,-81.525,-177.524,10.756,149.513
C05147=1114.076,329.785,-81.560,-177.521,10.758,149.513
C05148=1114.072,330.034,-81.593,-177.518,10.760,149.512
C05149=1114.068,330.281,-81.627,-177.515,10.763,149.512
C05150=1114.064,330.528,-81.661,-177.511,10.766,149.512
C05151=1114.060,330.777,-81.695,-177.508,10.768,149.512
C05152=1114.056,331.024,-81.729,-177.505,10.771,149.512
C05153=1114.052,331.271,-81.763,-177.502,10.773,149.512
C05154=1114.048,331.520,-81.797,-177.499,10.775,149.511
C05155=1114.044,331.767,-81.831,-177.496,10.777,149.511
C05156=1114.040,332.014,-81.865,-177.493,10.780,149.511
C05157=1114.036,332.263,-81.899,-177.490,10.783,149.511
C05158=1114.032,332.510,-81.933,-177.486,10.785,149.511
C05159=1114.029,332.758,-81.967,-177.483,10.788,149.510
C05160=1114.025,333.005,-82.001,-177.480,10.790,149.510
C05161=1114.020,333.253,-82.034,-177.477,10.793,149.510
C05162=1114.017,333.501,-82.069,-177.473,10.795,149.510
C05163=1114.013,333.748,-82.103,-177.470,10.798,149.510
C05164=1114.009,333.996,-82.137,-177.468,10.800,149.509
C05165=1114.006,334.243,-82.171,-177.464,10.802,149.509
C05166=1114.002,334.456,-82.200,-177.462,10.805,149.509
C05167=1113.998,334.667,-82.229,-177.459,10.807,149.509
C05168=1113.995,334.880,-82.259,-177.457,10.809,149.509
C05169=1113.992,335.092,-82.289,-177.453,10.811,149.509
C05170=1113.989,335.304,-82.318,-177.451,10.813,149.508
C05171=1113.984,335.516,-82.347,-177.448,10.816,149.508
C05172=1113.981,335.729,-82.376,-177.445,10.818,149.508
C05173=1113.978,335.941,-82.406,-177.443,10.819,149.508
C05174=1113.974,336.188,-82.440,-177.440,10.822,149.508
C05175=1113.970,336.436,-82.475,-177.436,10.824,149.508
C05176=1113.966,336.683,-82.508,-177.433,10.827,149.507
C05177=1113.962,336.931,-82.543,-177.430,10.829,149.507
C05178=1113.959,337.178,-82.577,-177.427,10.832,149.507
C05179=1113.955,337.426,-82.612,-177.424,10.835,149.507
C05180=1113.951,337.674,-82.646,-177.420,10.837,149.507
C05181=1113.947,337.922,-82.681,-177.418,10.839,149.506
C05182=1113.943,338.169,-82.715,-177.415,10.842,149.506
C05183=1113.939,338.417,-82.749,-177.411,10.844,149.506
C05184=1113.934,338.664,-82.784,-177.408,10.846,149.506
C05185=1113.931,338.912,-82.818,-177.405,10.849,149.506
C05186=1113.927,339.160,-82.853,-177.402,10.852,149.505
C05187=1113.924,339.407,-82.888,-177.398,10.854,149.505
C05188=1113.919,339.654,-82.922,-177.395,10.857,149.505
C05189=1113.915,339.902,-82.957,-177.392,10.859,149.505
C05190=1113.911,340.149,-82.991,-177.389,10.862,149.505
C05191=1113.907,340.398,-83.026,-177.386,10.864,149.505
C05192=1113.903,340.645,-83.060,-177.382,10.867,149.504
C05193=1113.900,340.892,-83.095,-177.380,10.868,149.504
C05194=1113.895,341.140,-83.129,-177.376,10.871,149.504
C05195=1113.891,341.388,-83.164,-177.373,10.874,149.504
C05196=1113.888,341.635,-83.198,-177.370,10.876,149.503
C05197=1113.884,341.882,-83.234,-177.367,10.879,149.503
C05198=1113.879,342.130,-83.268,-177.363,10.881,149.503
C05199=1113.876,342.378,-83.302,-177.360,10.884,149.503
C05200=1113.872,342.626,-83.337,-177.357,10.886,149.503
C05201=1113.868,342.872,-83.372,-177.354,10.889,149.503
C05202=1113.864,343.121,-83.407,-177.351,10.891,149.502
C05203=1113.860,343.368,-83.441,-177.347,10.894,149.502
C05204=1113.856,343.615,-83.477,-177.345,10.896,149.502
C05205=1113.852,343.863,-83.511,-177.342,10.898,149.502
C05206=1113.848,344.110,-83.547,-177.338,10.901,149.502
C05207=1113.845,344.358,-83.581,-177.335,10.903,149.501
C05208=1113.840,344.605,-83.615,-177.332,10.905,149.501
C05209=1113.837,344.853,-83.651,-177.328,10.908,149.501
C05210=1113.833,345.101,-83.686,-177.325,10.911,149.501
C05211=1113.828,345.348,-83.721,-177.322,10.913,149.501
C05212=1113.825,345.596,-83.755,-177.319,10.916,149.500
C05213=1113.822,345.843,-83.791,-177.316,10.918,149.500
C05214=1113.817,346.090,-83.825,-177.312,10.921,149.500
C05215=1113.813,346.338,-83.861,-177.310,10.923,149.500
C05216=1113.809,346.586,-83.896,-177.307,10.925,149.500
C05217=1113.805,346.833,-83.931,-177.303,10.928,149.499
C05218=1113.802,347.080,-83.966,-177.300,10.930,149.499
C05219=1113.798,347.328,-84.000,-177.297,10.932,149.499
C05220=1113.794,347.575,-84.036,-177.293,10.935,149.499
C05221=1113.790,347.823,-84.071,-177.290,10.938,149.499
C05222=1113.787,348.035,-84.101,-177.288,10.939,149.498
C05223=1113.783,348.247,-84.131,-177.284,10.942,149.498
C05224=1113.780,348.459,-84.161,-177.282,10.944,149.498
C05225=1113.777,348.671,-84.191,-177.279,10.946,149.498
C05226=1113.773,348.883,-84.222,-177.277,10.948,149.498
C05227=1113.770,349.095,-84.251,-177.274,10.950,149.497
C05228=1113.767,349.307,-84.282,-177.271,10.952,149.497
C05229=1113.763,349.520,-84.312,-177.268,10.954,149.497
C05230=1113.760,349.767,-84.347,-177.265,10.957,149.497
C05231=1113.755,350.014,-84.383,-177.262,10.959,149.497
C05232=1113.751,350.262,-84.418,-177.258,10.962,149.496
C05233=1113.748,350.509,-84.453,-177.255,10.964,149.496
C05234=1113.744,350.757,-84.489,-177.252,10.967,149.496
C05235=1113.740,351.004,-84.524,-177.248,10.969,149.496
C05236=1113.736,351.251,-84.559,-177.245,10.972,149.496
C05237=1113.732,351.499,-84.594,-177.242,10.974,149.495
C05238=1113.728,351.747,-84.630,-177.239,10.977,149.495
C05239=1113.724,351.994,-84.665,-177.235,10.979,149.495
C05240=1113.721,352.241,-84.700,-177.232,10.982,149.495
C05241=1113.717,352.489,-84.736,-177.229,10.984,149.494
C05242=1113.713,352.736,-84.772,-177.224,10.987,149.494
C05243=1113.710,352.984,-84.807,-177.221,10.989,149.494
C05244=1113.706,353.231,-84.843,-177.218,10.992,149.494
C05245=1113.702,353.478,-84.878,-177.214,10.994,149.493
C05246=1113.698,353.726,-84.913,-177.211,10.997,149.493
C05247=1113.694,353.973,-84.949,-177.208,10.999,149.493
C05248=1113.691,354.221,-84.984,-177.204,11.002,149.493
C05249=1113.686,354.468,-85.021,-177.201,11.004,149.493
C05250=1113.683,354.716,-85.056,-177.198,11.007,149.492
C05251=1113.678,354.963,-85.091,-177.194,11.009,149.492
C05252=1113.675,355.210,-85.127,-177.191,11.011,149.492
C05253=1113.671,355.458,-85.162,-177.187,11.014,149.491
C05254=1113.667,355.705,-85.198,-177.184,11.016,149.491
C05255=1113.664,355.953,-85.234,-177.181,11.019,149.491
C05256=1113.659,356.200,-85.270,-177.178,11.021,149.491
C05257=1113.656,356.448,-85.305,-177.174,11.023,149.490
C05258=1113.652,356.695,-85.341,-177.171,11.026,149.490
C05259=1113.649,356.942,-85.377,-177.167,11.028,149.490
C05260=1113.644,357.189,-85.412,-177.164,11.031,149.490
C05261=1113.640,357.437,-85.448,-177.161,11.033,149.490
C05262=1113.636,357.684,-85.484,-177.157,11.036,149.489
C05263=1113.633,357.932,-85.519,-177.154,11.038,149.489
C05264=1113.629,358.179,-85.556,-177.150,11.040,149.489
C05265=1113.625,358.427,-85.592,-177.147,11.043,149.488
C05266=1113.621,358.674,-85.627,-177.144,11.045,149.488
C05267=1113.618,358.921,-85.664,-177.140,11.048,149.488
C05268=1113.614,359.168,-85.699,-177.137,11.050,149.488
C05269=1113.610,359.416,-85.735,-177.133,11.052,149.487
C05270=1113.606,359.664,-85.771,-177.130,11.055,149.487
C05271=1113.603,359.911,-85.807,-177.127,11.057,149.487
C05272=1113.598,360.158,-85.843,-177.123,11.060,149.487
C05273=1113.595,360.405,-85.880,-177.120,11.062,149.486
C05274=1113.591,360.653,-85.915,-177.116,11.064,149.486
C05275=1113.587,360.901,-85.951,-177.113,11.067,149.486
C05276=1113.584,361.148,-85.988,-177.110,11.069,149.486
C05277=1113.580,361.395,-86.023,-177.107,11.072,149.486
C05278=1113.576,361.607,-86.054,-177.104,11.073,149.485
C05279=1113.573,361.818,-86.086,-177.101,11.076,149.485
C05280=1113.571,362.031,-86.116,-177.098,11.077,149.485
C05281=1113.567,362.243,-86.147,-177.095,11.079,149.485
C05282=1113.563,362.455,-86.178,-177.092,11.082,149.484
C05283=1113.560,362.666,-86.209,-177.089,11.083,149.484
C05284=1113.558,362.878,-86.240,-177.086,11.086,149.484
C05285=1113.554,363.090,-86.271,-177.083,11.087,149.484
C05286=1113.550,363.338,-86.307,-177.080,11.090,149.483
C05287=1113.546,363.585,-86.344,-177.077,11.092,149.483
C05288=1113.543,363.832,-86.380,-177.073,11.095,149.483
C05289=1113.539,364.080,-86.416,-177.070,11.097,149.483
C05290=1113.535,364.326,-86.452,-177.066,11.099,149.482
C05291=1113.531,364.574,-86.489,-177.063,11.102,149.482
C05292=1113.527,364.821,-86.525,-177.060,11.104,149.482
C05293=1113.523,365.068,-86.562,-177.056,11.107,149.482
C05294=1113.520,365.316,-86.597,-177.053,11.109,149.481
C05295=1113.516,365.564,-86.634,-177.049,11.112,149.481
C05296=1113.513,365.811,-86.671,-177.046,11.114,149.481
C05297=1113.509,366.058,-86.708,-177.043,11.116,149.481
C05298=1113.505,366.305,-86.743,-177.040,11.119,149.480
C05299=1113.501,366.552,-86.780,-177.036,11.121,149.480
C05300=1113.497,366.800,-86.817,-177.033,11.124,149.480
C05301=1113.494,367.046,-86.853,-177.029,11.126,149.480
C05302=1113.489,367.294,-86.889,-177.027,11.128,149.479
C05303=1113.486,367.542,-86.926,-177.023,11.130,149.479
C05304=1113.482,367.789,-86.963,-177.020,11.133,149.479
C05305=1113.478,368.036,-87.000,-177.017,11.135,149.479
C05306=1113.475,368.283,-87.036,-177.013,11.137,149.478
C05307=1113.470,368.531,-87.072,-177.010,11.140,149.478
C05308=1113.467,368.778,-87.108,-177.006,11.142,149.478
C05309=1113.463,369.025,-87.145,-177.003,11.145,149.478
C05310=1113.459,369.273,-87.182,-177.000,11.147,149.478
C05311=1113.456,369.520,-87.219,-176.996,11.150,149.477
C05312=1113.452,369.767,-87.255,-176.993,11.152,149.477
C05313=1113.448,370.014,-87.292,-176.989,11.154,149.477
C05314=1113.445,370.261,-87.329,-176.986,11.157,149.477
C05315=1113.441,370.509,-87.366,-176.983,11.159,149.476
C05316=1113.437,370.756,-87.403,-176.980,11.162,149.476
C05317=1113.433,371.003,-87.440,-176.976,11.164,149.476
C05318=1113.430,371.250,-87.476,-176.973,11.167,149.476
C05319=1113.426,371.498,-87.513,-176.970,11.169,149.475
C05320=1113.422,371.745,-87.550,-176.966,11.172,149.475
C05321=1113.419,371.992,-87.586,-176.963,11.174,149.475
C05322=1113.414,372.239,-87.623,-176.960,11.177,149.475
C05323=1113.411,372.487,-87.660,-176.956,11.179,149.474
C05324=1113.407,372.734,-87.697,-176.953,11.181,149.474
C05325=1113.403,372.982,-87.734,-176.949,11.184,149.474
C05326=1113.400,373.228,-87.771,-176.946,11.186,149.474
C05327=1113.396,373.476,-87.808,-176.943,11.189,149.474
C05328=1113.392,373.723,-87.845,-176.940,11.191,149.473
C05329=1113.388,373.970,-87.882,-176.936,11.194,149.473
C05330=1113.384,374.217,-87.919,-176.933,11.196,149.473
C05331=1113.382,374.464,-87.956,-176.930,11.199,149.473
C05332=1113.377,374.712,-87.993,-176.926,11.201,149.473
C05333=1113.373,374.959,-88.030,-176.923,11.204,149.472
C05334=1113.371,375.171,-88.062,-176.921,11.206,149.472
C05335=1113.367,375.382,-88.093,-176.918,11.208,149.472
C05336=1113.364,375.594,-88.126,-176.915,11.210,149.472
C05337=1113.360,375.806,-88.158,-176.912,11.213,149.472
C05338=1113.358,376.018,-88.190,-176.909,11.214,149.472
C05339=1113.354,376.229,-88.221,-176.906,11.217,149.472
C05340=1113.351,376.441,-88.252,-176.904,11.219,149.471
C05341=1113.348,376.653,-88.284,-176.901,11.221,149.471
C05342=1113.344,376.900,-88.322,-176.897,11.224,149.471
C05343=1113.341,377.147,-88.359,-176.894,11.226,149.471
C05344=1113.337,377.394,-88.396,-176.891,11.229,149.471
C05345=1113.333,377.641,-88.433,-176.888,11.232,149.471
C05346=1113.329,377.889,-88.471,-176.884,11.234,149.470
C05347=1113.326,378.136,-88.508,-176.881,11.237,149.470
C05348=1113.321,378.383,-88.545,-176.878,11.239,149.470
C05349=1113.318,378.630,-88.583,-176.874,11.242,149.470
C05350=1113.314,378.877,-88.620,-176.871,11.244,149.470
C05351=1113.310,379.124,-88.657,-176.868,11.247,149.470
C05352=1113.307,379.372,-88.695,-176.865,11.249,149.469
C05353=1113.303,379.618,-88.732,-176.862,11.252,149.469
C05354=1113.300,379.866,-88.769,-176.858,11.254,149.469
C05355=1113.296,380.113,-88.807,-176.856,11.257,149.469
C05356=1113.292,380.361,-88.844,-176.852,11.260,149.469
C05357=1113.289,380.607,-88.882,-176.849,11.262,149.469
C05358=1113.285,380.854,-88.919,-176.846,11.265,149.469
C05359=1113.281,381.102,-88.957,-176.843,11.267,149.468
C05360=1113.277,381.348,-88.994,-176.839,11.270,149.468
C05361=1113.274,381.596,-89.033,-176.837,11.273,149.468
C05362=1113.269,381.843,-89.070,-176.833,11.276,149.468
C05363=1113.266,382.090,-89.107,-176.829,11.278,149.468
C05364=1113.262,382.337,-89.145,-176.826,11.281,149.468
C05365=1113.259,382.585,-89.182,-176.823,11.284,149.468
C05366=1113.255,382.831,-89.220,-176.820,11.286,149.467
C05367=1113.252,383.079,-89.258,-176.817,11.289,149.467
C05368=1113.247,383.326,-89.295,-176.814,11.292,149.467
C05369=1113.244,383.573,-89.333,-176.811,11.294,149.467
C05370=1113.240,383.820,-89.371,-176.808,11.296,149.467
C05371=1113.237,384.067,-89.409,-176.806,11.299,149.467
C05372=1113.233,384.314,-89.446,-176.803,11.301,149.467
C05373=1113.230,384.562,-89.483,-176.800,11.304,149.467
C05374=1113.225,384.809,-89.522,-176.798,11.306,149.467
C05375=1113.222,385.056,-89.560,-176.795,11.309,149.467
C05376=1113.218,385.302,-89.597,-176.792,11.312,149.467
C05377=1113.215,385.550,-89.635,-176.791,11.314,149.467
C05378=1113.211,385.796,-89.673,-176.788,11.317,149.467
C05379=1113.207,386.044,-89.711,-176.785,11.319,149.467
C05380=1113.203,386.291,-89.748,-176.782,11.322,149.467
C05381=1113.200,386.538,-89.786,-176.780,11.325,149.467
C05382=1113.197,386.786,-89.824,-176.778,11.327,149.467
C05383=1113.192,387.033,-89.862,-176.775,11.330,149.467
C05384=1113.189,387.280,-89.900,-176.772,11.333,149.467
C05385=1113.185,387.526,-89.938,-176.770,11.335,149.467
C05386=1113.182,387.774,-89.976,-176.768,11.338,149.468
C05387=1113.178,388.020,-90.014,-176.765,11.341,149.468
C05388=1113.174,388.268,-90.052,-176.762,11.344,149.468
C05389=1113.171,388.515,-90.090,-176.760,11.346,149.468
C05390=1113.167,388.726,-90.123,-176.757,11.349,149.468
C05391=1113.165,388.938,-90.155,-176.755,11.352,149.468
C05392=1113.162,389.150,-90.188,-176.754,11.354,149.468
C05393=1113.159,389.360,-90.220,-176.752,11.356,149.468
C05394=1113.155,389.573,-90.253,-176.749,11.359,149.468
C05395=1113.153,389.784,-90.285,-176.747,11.361,149.468
C05396=1113.149,389.996,-90.318,-176.745,11.364,149.469
C05397=1113.146,390.207,-90.350,-176.743,11.366,149.469
C05398=1113.142,390.454,-90.389,-176.741,11.369,149.469
C05399=1113.138,390.701,-90.427,-176.738,11.372,149.469
C05400=1113.135,390.949,-90.464,-176.736,11.376,149.469
C05401=1113.131,391.195,-90.503,-176.733,11.379,149.469
C05402=1113.128,391.442,-90.541,-176.731,11.382,149.470
C05403=1113.124,391.690,-90.580,-176.728,11.385,149.470
C05404=1113.120,391.936,-90.617,-176.726,11.388,149.470
C05405=1113.117,392.184,-90.655,-176.724,11.392,149.470
C05406=1113.113,392.431,-90.695,-176.721,11.395,149.471
C05407=1113.110,392.677,-90.732,-176.719,11.398,149.471
C05408=1113.106,392.925,-90.771,-176.716,11.401,149.471
C05409=1113.102,393.172,-90.809,-176.714,11.405,149.471
C05410=1113.098,393.418,-90.847,-176.711,11.408,149.471
C05411=1113.095,393.666,-90.885,-176.709,11.411,149.472
C05412=1113.091,393.913,-90.924,-176.707,11.414,149.472
C05413=1113.088,394.160,-90.963,-176.705,11.418,149.472
C05414=1113.084,394.407,-91.001,-176.702,11.421,149.473
C05415=1113.080,394.654,-91.039,-176.700,11.424,149.473
C05416=1113.077,394.901,-91.078,-176.697,11.429,149.473
C05417=1113.073,395.147,-91.116,-176.695,11.432,149.474
C05418=1113.069,395.395,-91.154,-176.693,11.435,149.474
C05419=1113.066,395.642,-91.193,-176.691,11.439,149.474
C05420=1113.062,395.889,-91.231,-176.689,11.442,149.475
C05421=1113.059,396.135,-91.270,-176.687,11.446,149.475
C05422=1113.055,396.383,-91.308,-176.684,11.450,149.475
C05423=1113.052,396.629,-91.347,-176.682,11.453,149.476
C05424=1113.048,396.877,-91.385,-176.680,11.457,149.476
C05425=1113.044,397.123,-91.424,-176.677,11.461,149.477
C05426=1113.041,397.371,-91.462,-176.675,11.465,149.477
C05427=1113.037,397.618,-91.501,-176.673,11.468,149.478
C05428=1113.034,397.865,-91.539,-176.671,11.472,149.478
C05429=1113.030,398.111,-91.578,-176.668,11.476,149.478
C05430=1113.026,398.359,-91.617,-176.666,11.480,149.479
C05431=1113.023,398.605,-91.655,-176.664,11.484,149.479
C05432=1113.019,398.853,-91.694,-176.662,11.488,149.480
C05433=1113.015,399.100,-91.733,-176.660,11.492,149.480
C05434=1113.012,399.346,-91.771,-176.657,11.496,149.481
C05435=1113.008,399.593,-91.810,-176.655,11.500,149.481
C05436=1113.004,399.840,-91.849,-176.653,11.504,149.482
C05437=1113.001,400.088,-91.887,-176.651,11.508,149.482
C05438=1112.998,400.335,-91.926,-176.649,11.512,149.483
C05439=1112.994,400.582,-91.966,-176.647,11.516,149.483
C05440=1112.990,400.827,-92.004,-176.645,11.521,149.484
C05441=1112.986,401.075,-92.043,-176.643,11.524,149.485
C05442=1112.983,401.322,-92.082,-176.641,11.529,149.485
C05443=1112.980,401.569,-92.120,-176.638,11.534,149.486
C05444=1112.976,401.816,-92.159,-176.636,11.537,149.486
C05445=1112.972,402.063,-92.198,-176.634,11.542,149.487
C05446=1112.969,402.275,-92.232,-176.632,11.546,149.487
C05447=1112.966,402.485,-92.265,-176.631,11.550,149.488
C05448=1112.963,402.697,-92.298,-176.629,11.553,149.489
C05449=1112.960,402.908,-92.331,-176.627,11.557,149.489
C05450=1112.957,403.119,-92.365,-176.625,11.561,149.490
C05451=1112.954,403.331,-92.398,-176.624,11.565,149.490
C05452=1112.951,403.543,-92.432,-176.622,11.568,149.491
C05453=1112.948,403.755,-92.465,-176.620,11.572,149.491
